(* CODESYS project Rasi_feeds_batching2.project

Project tree, tasks and I/O mapping:
  PLC_AC500_V3 : PM5032-T-ETH, ABB AG, order no. 1SAP123400R0x72, version 3.7.0.0
    application Application
      libraries: ModbusRtu, * (ABB); Util, * (System)
      task Task (cyclic, interval t#10ms, priority 14, watchdog t#20ms x 1) calls batching14
      CheckConfigurationObject
      Diagnosis/
        text list Diag_IO_Bus
        text list Diag_V3_PLC
      global variables GVL
      function block Auto_Batching_V14 [ST]
      function block Semi_Auto_Batching_V14 [ST]
      program batching14 [FBD]
      function block FB_Samyak_Multi [ST]
      function block FB_Samyak_Control [ST]
    OnBoard_IO : 12DI/8DO-T/2DC, ABB AG, version 3.7.0.0
        input  E_Stop_DI : BOOL  // Fast inputs DI0-DI3.Digital input DI0
        input  Run_PB : BOOL  // Fast inputs DI0-DI3.Digital input DI1
        unmapped channels: Fast inputs DI0-DI3, Fast inputs DI4-DI7, Standard inputs DI8-DI11, Digital inputs - Transistor, Fast outputs DO0-DO3, Fast outputs DO4-DO7, Digital outputs - Transistor
    IO_Bus : I/O-Bus, ABB AG, version 3.7.0.0
    Interfaces : Interfaces, ABB AG, version 3.7.0.0
      TA5142_RS485I : TA5142-RS485I, ABB AG, order no. 1SAP187300R0x02, version 3.7.0.0
        Modbus_RTU_Client : Modbus RTU Client, ABB AG, version 3.7.0.0
      OptionSlot_2
      Ethernet : Ethernet, ABB AG, version 3.7.0.0
        ETH1 : IP Settings, ABB AG, version 3.7.0.0
          NetConfig : NetConfig, ABB AG, version 3.7.0.0
          Modbus_TCP_IP_Server : Modbus TCP/IP Server, ABB AG, version 3.7.0.0
        Protocols : Client Protocols, ABB AG, version 3.7.0.0
    OnBoard_RTC : OnBoard RTC, ABB AG, version 3.7.0.0
  text list GlobalTextList
*)

// PLC_AC500_V3/Application/GVL
{attribute 'qualified_only'}
VAR_GLOBAL
    Recipe_Weights AT %MD100 : ARRAY[1..20] OF REAL;
	Auto_Bin_Material_Mapping AT %MW50: ARRAY[1..6] OF INT;
	Semi_Auto_Bin_Material_Mapping AT %MW60: ARRAY[1..10] OF INT;
	Auto_Coarse_To_Fine_speed AT %MD120: ARRAY[1..6] OF REAL := [1.0,1.0,1.0,1.0,1.0,1.0];
	Semi_Auto_Coarse_To_Fine_speed AT %MD130: ARRAY[1..10] OF REAL := [1.0,1.0,1.0,1.0,1.0,1.0,1.0,1.0,1.0,1.0];
	Auto_Bin_Tolerance AT %MD150: ARRAY[1..6] OF REAL;
	Semi_Auto_Bin_Tolerance AT %MD160: ARRAY[1..10] OF REAL;
	Start_Button AT %MX2.0: BOOL;
	E_Stop_Active AT %MX2.1: BOOL;
	Reset AT %MX2.3: BOOL;
	Next_Cycle_Start AT %MX2.4: BOOL;               // Command pulse/signal to start next batch cycle after hoppers are emptied
	Auto_Active_Mat AT %MW70: INT;
	Auto_Active_Bin AT %MW71: INT;
	Semi_Auto_Active_Mat AT %MW72: INT;
	Semi_Auto_Active_Bin AT %MW73: INT;
	Target_Batch_Cycles AT %MW74: INT := 1;
	Current_Batch_Cycle AT %MW75: INT;
	Completed_Batch_Cycles AT %MW79: INT;
	Error_Code AT %MW76: INT;
	Run AT %MX2.5 : BOOL;
	load_cell_auto AT %MD174 : REAL;
	load_cell_semi_auto AT %MD175 : REAL;
	Auto_Initial_Tolerance AT %MD176 : REAL := 5.0;
	Semi_Auto_Initial_Tolerance AT %MD178 : REAL := 5.0;
	Empty_Weight_Limit AT %MD186 : REAL := 5.0;     // Maximum scale weight limit (kg) to qualify scale as empty before starting next cycle
	Auto_Total_Target_Weight AT %MD170 : REAL;
	Semi_Auto_Total_Target_Weight AT %MD171 : REAL;
	Auto_Material_Count AT %MW77: INT;
	Semi_Auto_Material_Count AT %MW78 : INT;
	Auto_Current_Step AT %MW80 : INT;
	Semi_Auto_Current_Step AT %MW81 : INT;
	Auto_Active_Target_Weight AT %MD220 : REAL;
	Semi_Auto_Active_Target_Weight AT %MD224 : REAL;
	Auto_Active_Live_Weight AT %MD172 : REAL;
	Semi_Auto_Active_Live_Weight AT %MD173 : REAL;
	Auto_Excess_Allowed AT %MX2.6 : BOOL;
	Semi_Auto_Excess_Allowed AT %MX2.9 : BOOL;
	Auto_Excess_Alarm AT %MX2.7 : BOOL;
	Semi_Auto_Excess_Alarm AT %MX2.8 : BOOL;
	Auto_Inter_Bin_Delay AT %MD190 : TIME;
	Semi_Auto_Inter_Bin_Delay AT %MD194 : TIME;
	Auto_Sequence_Complete AT %MX3.0 : BOOL;
	Semi_Auto_Sequence_Complete AT %MX3.1 : BOOL;
	All_Cycles_Complete AT %MX3.2 : BOOL;           // Master flag: TRUE when all target batch cycles have completed
	Auto_Status_Message : STRING(80);
	Semi_Auto_Status_Message : STRING(80);
	
	(* 8 Process Output and Weight Arrays *)
	Auto_Bin : ARRAY[1..6] OF BOOL;
	auto_bin_cutoff : ARRAY[1..6] OF BOOL;
	auto_bin_motor : ARRAY[1..6] OF BOOL;
	Semi_Auto_Bin : ARRAY[1..10] OF BOOL;
	semi_auto_bin_cutoff : ARRAY[1..10] OF BOOL;
	semi_auto_bin_motor : ARRAY[1..10] OF BOOL;
	Auto_Weights : ARRAY[1..6] OF REAL;
	Semi_Auto_Weights : ARRAY[1..10] OF REAL;
END_VAR

// PLC_AC500_V3/Application/batching14
PROGRAM batching14
VAR
	Auto_Ctrl: Auto_Batching_V14;
	Semi_Auto_Ctrl: Semi_Auto_Batching_V14;
	Auto_Complete: BOOL;
	Semi_Auto_Complete: BOOL;
	Auto_Err: INT;
	Auto_Msg: STRING;
	Semi_Auto_Err: INT;
	Semi_Auto_Msg: STRING;
	AutoBatchScale: MODRTUMAST;
	ModEnabler: BLINK;
	SamyakRaw: ARRAY[0..1] OF DINT;
	AutBatchRaw: ARRAY[0..1] OF DINT;
	SemAutoScale: MODRTUMAST;
	SemiAutoScaleRaw: ARRAY[0..1] OF DINT;
	AutoBatchSamyak: REAL;
	FB_Samyak_Multi_1: FB_Samyak_Multi;
	
	FB_Samyak_Control_1: FB_Samyak_Control;
	Run_PB_1: BOOL;
	Next_Cycle_Start: BOOL;
END_VAR

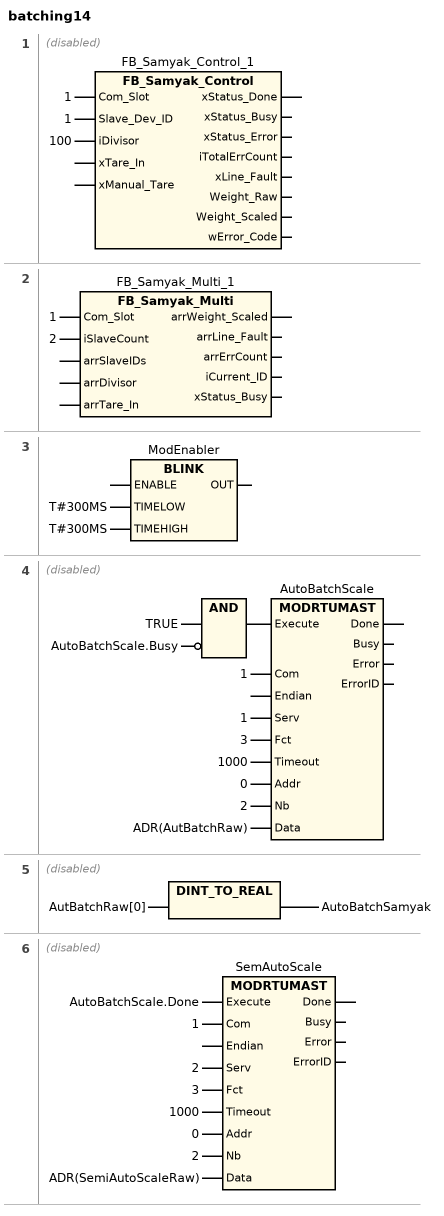
// NETWORK 1 (disabled)
// FB_Samyak_Control_1(Com_Slot := 1, Slave_Dev_ID := 1, iDivisor := 100); // FB_Samyak_Control

// NETWORK 2
FB_Samyak_Multi_1(Com_Slot := 1, iSlaveCount := 2); // FB_Samyak_Multi

// NETWORK 3
ModEnabler(TIMELOW := T#300MS, TIMEHIGH := T#300MS); // BLINK

// NETWORK 4 (disabled)
// AutoBatchScale(
//     Execute := TRUE AND NOT AutoBatchScale.Busy,
//     Com := 1,
//     Serv := 1,
//     Fct := 3,
//     Timeout := 1000,
//     Addr := 0,
//     Nb := 2,
//     Data := ADR(AutBatchRaw)); // MODRTUMAST

// NETWORK 5 (disabled)
// AutoBatchSamyak := DINT_TO_REAL(AutBatchRaw[0]);

// NETWORK 6 (disabled)
// SemAutoScale(
//     Execute := AutoBatchScale.Done,
//     Com := 1,
//     Serv := 2,
//     Fct := 3,
//     Timeout := 1000,
//     Addr := 0,
//     Nb := 2,
//     Data := ADR(SemiAutoScaleRaw)); // MODRTUMAST

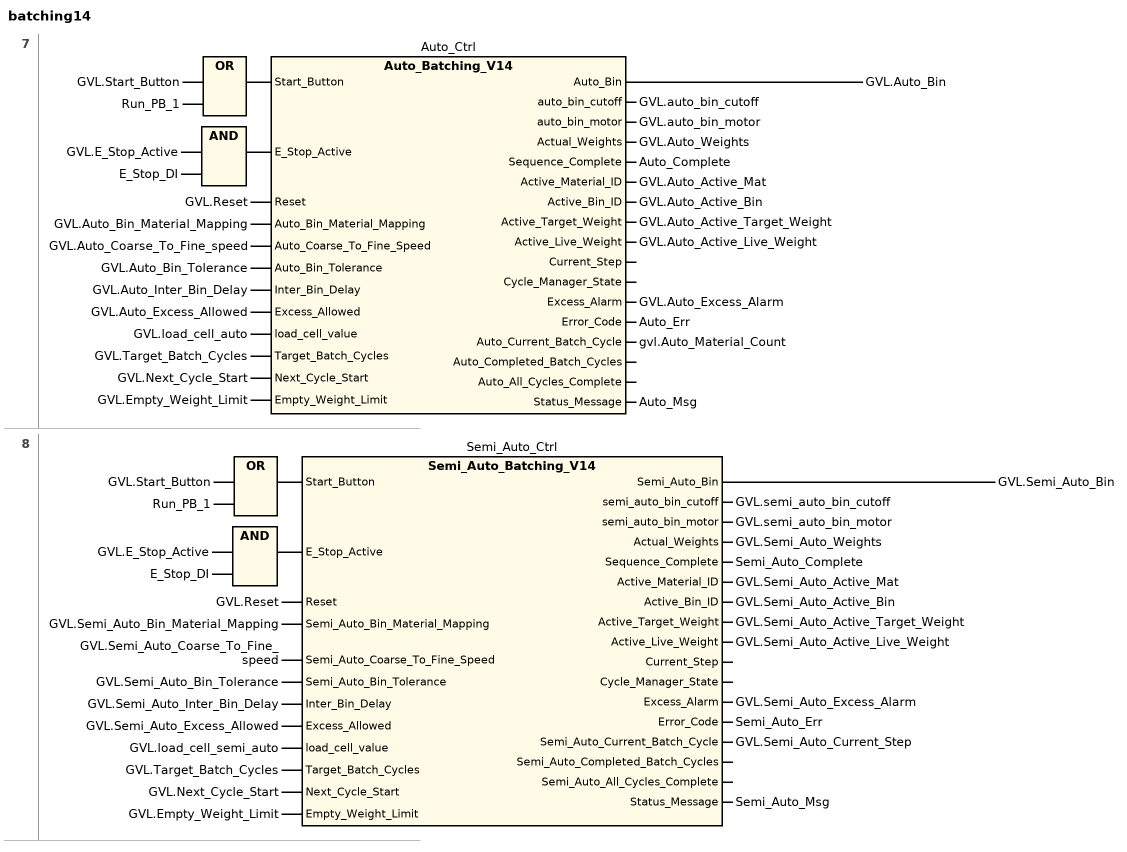
// NETWORK 7
Auto_Ctrl(
    Start_Button := GVL.Start_Button OR Run_PB_1,
    E_Stop_Active := GVL.E_Stop_Active AND E_Stop_DI,
    Reset := GVL.Reset,
    Auto_Bin_Material_Mapping := GVL.Auto_Bin_Material_Mapping,
    Auto_Coarse_To_Fine_Speed := GVL.Auto_Coarse_To_Fine_speed,
    Auto_Bin_Tolerance := GVL.Auto_Bin_Tolerance,
    Inter_Bin_Delay := GVL.Auto_Inter_Bin_Delay,
    Excess_Allowed := GVL.Auto_Excess_Allowed,
    load_cell_value := GVL.load_cell_auto,
    Target_Batch_Cycles := GVL.Target_Batch_Cycles,
    Next_Cycle_Start := GVL.Next_Cycle_Start,
    Empty_Weight_Limit := GVL.Empty_Weight_Limit,
    auto_bin_cutoff => GVL.auto_bin_cutoff,
    auto_bin_motor => GVL.auto_bin_motor,
    Actual_Weights => GVL.Auto_Weights,
    Sequence_Complete => Auto_Complete,
    Active_Material_ID => GVL.Auto_Active_Mat,
    Active_Bin_ID => GVL.Auto_Active_Bin,
    Active_Target_Weight => GVL.Auto_Active_Target_Weight,
    Active_Live_Weight => GVL.Auto_Active_Live_Weight,
    Excess_Alarm => GVL.Auto_Excess_Alarm,
    Error_Code => Auto_Err,
    Auto_Current_Batch_Cycle => gvl.Auto_Material_Count,
    Status_Message => Auto_Msg); // Auto_Batching_V14
GVL.Auto_Bin := Auto_Ctrl.Auto_Bin;

// NETWORK 8
Semi_Auto_Ctrl(
    Start_Button := GVL.Start_Button OR Run_PB_1,
    E_Stop_Active := GVL.E_Stop_Active AND E_Stop_DI,
    Reset := GVL.Reset,
    Semi_Auto_Bin_Material_Mapping := GVL.Semi_Auto_Bin_Material_Mapping,
    Semi_Auto_Coarse_To_Fine_Speed := GVL.Semi_Auto_Coarse_To_Fine_speed,
    Semi_Auto_Bin_Tolerance := GVL.Semi_Auto_Bin_Tolerance,
    Inter_Bin_Delay := GVL.Semi_Auto_Inter_Bin_Delay,
    Excess_Allowed := GVL.Semi_Auto_Excess_Allowed,
    load_cell_value := GVL.load_cell_semi_auto,
    Target_Batch_Cycles := GVL.Target_Batch_Cycles,
    Next_Cycle_Start := GVL.Next_Cycle_Start,
    Empty_Weight_Limit := GVL.Empty_Weight_Limit,
    semi_auto_bin_cutoff => GVL.semi_auto_bin_cutoff,
    semi_auto_bin_motor => GVL.semi_auto_bin_motor,
    Actual_Weights => GVL.Semi_Auto_Weights,
    Sequence_Complete => Semi_Auto_Complete,
    Active_Material_ID => GVL.Semi_Auto_Active_Mat,
    Active_Bin_ID => GVL.Semi_Auto_Active_Bin,
    Active_Target_Weight => GVL.Semi_Auto_Active_Target_Weight,
    Active_Live_Weight => GVL.Semi_Auto_Active_Live_Weight,
    Excess_Alarm => GVL.Semi_Auto_Excess_Alarm,
    Error_Code => Semi_Auto_Err,
    Semi_Auto_Current_Batch_Cycle => GVL.Semi_Auto_Current_Step,
    Status_Message => Semi_Auto_Msg); // Semi_Auto_Batching_V14
GVL.Semi_Auto_Bin := Semi_Auto_Ctrl.Semi_Auto_Bin;

END_PROGRAM

// PLC_AC500_V3/Application/FB_Samyak_Control
FUNCTION_BLOCK FB_Samyak_Control
VAR_INPUT
    Com_Slot      : BYTE := 1;     (* PLC COM port *)
    Slave_Dev_ID  : BYTE := 1;     (* Samyak slave ID *)
    iDivisor      : REAL := 10.0;  (* Scale factor: Weight_Scaled = Raw / iDivisor *)
    xTare_In      : BOOL;           (* Logic tare pulse *)
    xManual_Tare  : BOOL;           (* HMI/manual tare pulse *)
END_VAR

VAR_OUTPUT
    xStatus_Done   : BOOL;
    xStatus_Busy   : BOOL;
    xStatus_Error  : BOOL;
    iTotalErrCount : INT := 0;
    xLine_Fault    : BOOL;
    Weight_Raw     : DINT;
    Weight_Scaled  : REAL;
    wError_Code    : WORD; (* Check PLC & SAMYAK BaudRate, DevId, Parity; also check PLC serial port LED blink status and RS485 connection if error repeats *)
END_VAR

VAR
    fbRead         : ModRtuMast;
    fbTare         : ModRtuMast;
    iStep          : INT := 0;
    Samyak_Buffer  : ARRAY[0..17] OF WORD;
    wTareCommand   : WORD := 1;

    rtTareTrig     : R_TRIG;
    rtErrTrig      : R_TRIG;
    tStuckWatchdog : TON;
    tRecoveryTimer : TON;

    xTareReq       : BOOL := FALSE; (* Internal tare request latch *)
END_VAR


(* --- 1) Error Tracking + Auto Recovery --- *)
tStuckWatchdog(IN := (fbRead.Busy OR fbTare.Busy), PT := T#2000MS);

rtErrTrig(CLK := (fbRead.Error OR fbTare.Error));
IF rtErrTrig.Q THEN
    iTotalErrCount := iTotalErrCount + 1;
END_IF

IF fbRead.Done OR fbTare.Done THEN
    iTotalErrCount := 0;
    xLine_Fault := FALSE;
END_IF

IF iTotalErrCount >= 10 THEN
    xLine_Fault := TRUE;
END_IF

tRecoveryTimer(IN := xLine_Fault, PT := T#5S);
IF tRecoveryTimer.Q THEN
    iTotalErrCount := 0;
    xLine_Fault := FALSE;
END_IF

IF tStuckWatchdog.Q THEN
    iStep := 99;
END_IF

(* Capture tare request from either input pulse *)
rtTareTrig(CLK := xTare_In OR xManual_Tare);
IF rtTareTrig.Q THEN
    xTareReq := TRUE;
END_IF

(* --- 2) Modbus State Machine --- *)
CASE iStep OF

    0:  (* Continuous Read *)
        fbTare(Execute := FALSE);

        fbRead(
            Execute := NOT (fbRead.Done OR fbRead.Error OR fbRead.Busy)
                       AND NOT xTareReq
                       AND NOT xLine_Fault,
            COM     := Com_Slot,
            Serv    := Slave_Dev_ID,
            FCT     := 3,
            Addr    := 0,
            Nb      := 2,
            Data    := ADR(Samyak_Buffer[0]),
            Timeout := 400,
            Done    => xStatus_Done,
            Busy    => xStatus_Busy,
            Error   => xStatus_Error,
            ErrorID => wError_Code
        );

        IF xStatus_Done THEN
            Weight_Raw := TO_DINT(SHL(TO_DWORD(Samyak_Buffer[1]), 16) OR TO_DWORD(Samyak_Buffer[0]));
            Weight_Scaled := TO_REAL(Weight_Raw) / iDivisor;
        END_IF

        IF xTareReq THEN
            iStep := 1;
        END_IF

    1:  (* Port Release *)
        fbRead(Execute := FALSE);
        IF NOT fbRead.Busy THEN
            iStep := 2;
        END_IF

    2:  (* Execute Tare *)
        fbTare(
            Execute := TRUE,
            COM     := Com_Slot,
            Serv    := Slave_Dev_ID,
            FCT     := 6,
            Addr    := 16,
            Nb      := 1,
            Data    := ADR(wTareCommand),
            Timeout := 1000,
            Done    => xStatus_Done,
            Busy    => xStatus_Busy,
            Error   => xStatus_Error,
            ErrorID => wError_Code
        );

        IF fbTare.Done OR fbTare.Error THEN
            xTareReq := FALSE;
            iStep := 3;
        END_IF

    3:  (* Return to Read *)
        fbTare(Execute := FALSE);
        IF NOT fbTare.Busy THEN
            iStep := 0;
        END_IF

    99: (* Emergency Recovery *)
        fbRead(Execute := FALSE);
        fbTare(Execute := FALSE);

        IF NOT (fbRead.Busy OR fbTare.Busy) THEN
            iTotalErrCount := 0;
            iStep := 0;
        END_IF

END_CASE

END_FUNCTION_BLOCK

// PLC_AC500_V3/Application/FB_Samyak_Multi
//SAMYAK 4016 Multi Slave Unit Customised Block
//Note: This FB_Samyak_Multi name is impotrtant when you create new POU.

FUNCTION_BLOCK FB_Samyak_Multi
VAR_INPUT
    Com_Slot      : BYTE := 1;    (* Port Number *)
    iSlaveCount   : INT := 1;     (* How many slaves active: 1 to 4 *)
    arrSlaveIDs   : ARRAY[1..4] OF BYTE := [1, 2, 3, 4]; (* Unit IDs *)
    arrDivisor    : ARRAY[1..4] OF REAL := [10.0, 10.0, 10.0, 10.0]; (* Scaling per Unit *)
    arrTare_In    : ARRAY[1..4] OF BOOL; (* Individual Tare triggers *)
END_VAR

VAR_OUTPUT
    arrWeight_Scaled : ARRAY[1..4] OF REAL; (* Scaled result per unit *)
    arrLine_Fault    : ARRAY[1..4] OF BOOL; (* Fault status per unit *)
    arrErrCount      : ARRAY[1..4] OF INT;  (* Error count per unit *)
    iCurrent_ID      : BYTE;                (* Current ID being polled *)
    xStatus_Busy     : BOOL;                (* Overall Bus Busy *)
END_VAR

VAR
    (* Internal ModRtuMast Instances *)
    fbRead         : ModRtuMast;
    fbTare         : ModRtuMast;
    
    (* Polling Control *)
    iStep          : INT := 0;
    iIdx           : INT := 1;    (* Current Loop Index *)
    Samyak_Buffer  : ARRAY[0..17] OF WORD;
    wTareCommand   : WORD := 1;
    
    (* Unique Timer/Trigger Instances *)
    rtTareTrig     : R_TRIG;
    rtErrTrig      : R_TRIG;
    tWatchdog      : TON;
    tRecovery      : TON;
END_VAR



(* --- 1. INDIVIDUAL UNIT MONITORING --- *)
iCurrent_ID := arrSlaveIDs[iIdx]; 

(* Watchdog for Bus Hangs *)
tWatchdog(IN := (fbRead.Busy OR fbTare.Busy), PT := T#2000MS);
xStatus_Busy := fbRead.Busy OR fbTare.Busy;

(* Error Tracking for Current Index *)
rtErrTrig(CLK := (fbRead.Error OR fbTare.Error));
IF rtErrTrig.Q THEN
    arrErrCount[iIdx] := arrErrCount[iIdx] + 1;
END_IF

(* Reset on Success *)
IF fbRead.Done OR fbTare.Done THEN
    arrErrCount[iIdx] := 0;
    arrLine_Fault[iIdx] := FALSE;
END_IF

(* Line Fault Activation (10 errors) *)
IF arrErrCount[iIdx] >= 10 THEN
    arrLine_Fault[iIdx] := TRUE;
END_IF

(* Auto-Recovery pulse (5s) *)
tRecovery(IN := arrLine_Fault[iIdx], PT := T#5S);
IF tRecovery.Q THEN
    arrErrCount[iIdx] := 0;
    arrLine_Fault[iIdx] := FALSE;
END_IF

IF tWatchdog.Q THEN iStep := 99; END_IF

(* Check Tare for active slave *)
rtTareTrig(CLK := arrTare_In[iIdx]);

(* --- 2. SEQUENTIAL STATE MACHINE --- *)
CASE iStep OF
    
    0: (* READ CURRENT SLAVE *)
        fbTare(Execute := FALSE);
        fbRead(
            Execute := NOT (fbRead.Done OR fbRead.Error OR fbRead.Busy) 
                       AND NOT rtTareTrig.Q AND NOT arrLine_Fault[iIdx],
            COM     := Com_Slot,
            Serv    := arrSlaveIDs[iIdx],
            FCT     := 3, Addr := 0, Nb := 2, 
            Data    := ADR(Samyak_Buffer[0]), Timeout := 400
        );

        IF fbRead.Done THEN
            (* Scale weight using the array-based divisor for this specific index *)
            arrWeight_Scaled[iIdx] := TO_REAL(TO_DINT(SHL(TO_DWORD(Samyak_Buffer[1]), 16) OR TO_DWORD(Samyak_Buffer[0]))) / arrDivisor[iIdx];
            iStep := 10; (* Switch to next slave *)
        END_IF
        
        IF fbRead.Error THEN iStep := 10; END_IF (* Move on if error *)
        IF rtTareTrig.Q THEN iStep := 1; END_IF  (* Priority: Tare current unit *)

    1: (* PORT RELEASE *)
        fbRead(Execute := FALSE);
        IF NOT fbRead.Busy THEN iStep := 2; END_IF

    2: (* WRITE TARE FOR CURRENT SLAVE *)
        fbTare(
            Execute := TRUE,
            COM := Com_Slot, Serv := arrSlaveIDs[iIdx], 
            FCT := 6, Addr := 16, Nb := 1,
            Data := ADR(wTareCommand), Timeout := 1000
        );

        IF fbTare.Done OR fbTare.Error THEN
            arrTare_In[iIdx] := FALSE; (* Reset manual trigger *)
            iStep := 3;
        END_IF

    3: (* CLEANUP *)
        fbTare(Execute := FALSE);
        IF NOT fbTare.Busy THEN iStep := 10; END_IF

    10: (* INDEX ROTATION *)
        iIdx := iIdx + 1;
        IF iIdx > iSlaveCount THEN
            iIdx := 1; (* Back to first slave *)
        END_IF
        iStep := 0;

    99: (* EMERGENCY RESET *)
        fbRead(Execute := FALSE); fbTare(Execute := FALSE);
        IF NOT (fbRead.Busy OR fbTare.Busy) THEN iStep := 0; END_IF
        
END_CASE

END_FUNCTION_BLOCK

// PLC_AC500_V3/Application/Auto_Batching_V14
FUNCTION_BLOCK Auto_Batching_V14
VAR_INPUT
    Start_Button : BOOL;                            // Command pulse/signal to start or resume the auto batching sequence
    E_Stop_Active : BOOL;                           // Emergency Stop circuit status (NC contact: TRUE = Healthy/Run permitted, FALSE = E-Stop tripped)
    Reset : BOOL;                                   // System reset pulse (clears active steps, outputs, alarms, and error flags)
    Auto_Bin_Material_Mapping : ARRAY[1..6] OF INT; // Array mapping physical Silos 1..6 to Recipe Material IDs (1..20, 0 = Silo skipped)
    Auto_Coarse_To_Fine_Speed : ARRAY[1..6] OF REAL;// Weight offset threshold (kg) before target to transition from Coarse to Fine feeding
    Auto_Bin_Tolerance : ARRAY[1..6] OF REAL;       // Allowable weight tolerance window (±kg) around target weight for each silo
    Inter_Bin_Delay : TIME;                         // Settling delay duration after completing a bin before advancing to the next
    Excess_Allowed : BOOL;                          // Overfill handling policy: TRUE = proceed if target is exceeded, FALSE = raise alarm and halt
    load_cell_value : REAL;                         // Live gross weight input reading from the Auto scale load cell (kg)
    Target_Batch_Cycles : INT;                      // Target number of batch cycle repetitions configured from HMI (defaults to 1)
    Next_Cycle_Start : BOOL;                        // Command pulse/signal to start next batch cycle after hoppers are emptied
    Empty_Weight_Limit : REAL;                      // Maximum scale weight limit (kg) for scales to qualify as empty before starting next cycle
END_VAR
VAR_OUTPUT
    Auto_Bin : ARRAY[1..6] OF BOOL;                 // Coarse feeding valve / gate actuation command outputs for Silos 1..6
    auto_bin_cutoff : ARRAY[1..6] OF BOOL;          // Fine feeding valve / vibrator cutoff actuation command outputs for Silos 1..6
    auto_bin_motor : ARRAY[1..6] OF BOOL;           // Feeder / screw conveyor motor run commands for Silos 1..6
    Actual_Weights : ARRAY[1..6] OF REAL;           // Net material weight (kg) successfully dosed for each silo in the current cycle
    Sequence_Complete : BOOL;                       // Handshake flag: TRUE when all mapped Auto silos have completed dosing and settling
    Active_Material_ID : INT;                       // Recipe Material ID currently being dosed (1..20, 0 when idle/complete)
    Active_Bin_ID : INT;                            // Physical Silo index currently being dosed (1..6, 0 when idle/complete)
    Active_Target_Weight : REAL;                    // Target weight setpoint (kg) of the ingredient currently being dosed
    Active_Live_Weight : REAL;                      // Live net/tared weight (kg) accumulated into the scale for the active silo
    Current_Step : INT;                             // Real-time sequence step:
                                                    //   0  = Idle / Waiting for Start
                                                    //   1..6 = Dosing Silos 1..6 (feeding coarse/fine)
                                                    //   7  = Settling delay in progress
                                                    //   8  = Sequence complete
    Cycle_Manager_State : INT;                      // Master supervisory cycle manager state:
                                                    //   0  = System Idle / Stopped
                                                    //   1  = Running active batch cycle
                                                    //   4  = All target batch cycles completed successfully
                                                    //   5  = Paused between cycles (Cycle Hold active)
    Excess_Alarm : BOOL;                            // Overfill alarm: TRUE when dosed weight exceeds target + tolerance (with Excess_Allowed=FALSE)
    Error_Code : INT;                               // Fault diagnostic code:
                                                    //   0  = No Error / System Healthy
                                                    //   1  = Duplicate Material ID mapped across Auto and Semi-Auto
                                                    //   2  = Material index out of range (must be 1..20)
                                                    //   3  = Recipe weight is less than (Coarse_To_Fine_Speed + Tolerance)
                                                    //   4  = Initial scale tare error (scale not empty before start)
                                                    //   21 = Scale overload protection triggered (> 500 kg)
    Auto_Current_Batch_Cycle : INT;                     // Active batch cycle number currently processing (1..Target_Batch_Cycles)
    Auto_Completed_Batch_Cycles : INT;                  // Total number of batch cycle loops completed successfully
    Auto_All_Cycles_Complete : BOOL;                    // Master flag: TRUE when all Target_Batch_Cycles have finished
    Status_Message : STRING(80);                    // Real-time human-readable process status and diagnostic text message
END_VAR
VAR
    bin_last_weight : REAL;
    actual_bin : REAL;
    target_weight : REAL;
    cutoff_trigger_weight : REAL;
    min_tol_weight : REAL;
    max_tol_weight : REAL;
    Paused_By_EStop : BOOL;
    Effective_Delay : TIME;
    Mat_Idx : INT;
    i : INT;
    j : INT;
    Transition_Timer : TON;
    Completion_Timer : TON;
    Simulation_Mode : BOOL;
    Sim_Rate : REAL;
    Sim_Timer : TON;
    Start_Sim_Weight : REAL;
    Discharge_Active : BOOL;
    
    (* Master Cycle Manager & Supervisory states *)
    Internal_FB_Start : BOOL;
    Duplicate_Found : BOOL;
    Invalid_Material_Range : BOOL;
    Weight_Limit_Error : BOOL;
    eff_empty_limit : REAL;
    Next_Cycle_Last : BOOL;
    Next_Cycle_Rising : BOOL;
END_VAR


(* Auto Batching FB V14 with Full Diagnostics, Step Tracking, and Precise Status Reporting *)

Effective_Delay := Inter_Bin_Delay;
IF Effective_Delay = T#0S THEN
    Effective_Delay := T#2S;
END_IF;

(* Detect rising edge on Next_Cycle_Start trigger *)
Next_Cycle_Rising := (Next_Cycle_Start OR GVL.Next_Cycle_Start) AND NOT Next_Cycle_Last;
Next_Cycle_Last := (Next_Cycle_Start OR GVL.Next_Cycle_Start);

(* 1. RECIPE TOTALS & SUPERVISORY CONFIGURATION CHECKS *)
Duplicate_Found := FALSE;
Invalid_Material_Range := FALSE;
Weight_Limit_Error := FALSE;

GVL.Auto_Total_Target_Weight := 0.0;
GVL.Auto_Material_Count := 0;
FOR i := 1 TO 6 DO
    IF Auto_Bin_Material_Mapping[i] < 0 OR Auto_Bin_Material_Mapping[i] > 20 THEN
        Invalid_Material_Range := TRUE;
    END_IF;
    IF Auto_Bin_Material_Mapping[i] <> 0 AND Auto_Bin_Material_Mapping[i] <= 20 THEN
        FOR j := 1 TO 10 DO
            IF Auto_Bin_Material_Mapping[i] = GVL.Semi_Auto_Bin_Material_Mapping[j] THEN
                Duplicate_Found := TRUE;
            END_IF;
        END_FOR;
    END_IF;
    IF Auto_Bin_Material_Mapping[i] > 0 AND Auto_Bin_Material_Mapping[i] <= 20 THEN
        IF GVL.Recipe_Weights[Auto_Bin_Material_Mapping[i]] > 0.0 THEN
            GVL.Auto_Total_Target_Weight := GVL.Auto_Total_Target_Weight + GVL.Recipe_Weights[Auto_Bin_Material_Mapping[i]];
            GVL.Auto_Material_Count := GVL.Auto_Material_Count + 1;
            IF GVL.Recipe_Weights[Auto_Bin_Material_Mapping[i]] < (Auto_Coarse_To_Fine_Speed[i] + Auto_Bin_Tolerance[i]) THEN
                Weight_Limit_Error := TRUE;
            END_IF;
        END_IF;
    END_IF;
END_FOR;

IF Duplicate_Found THEN
    GVL.Error_Code := 1;
    Error_Code := 1;
    Status_Message := 'Error 1: Duplicate Material ID mapped in Auto and Semi-Auto!';
ELSIF Invalid_Material_Range THEN
    GVL.Error_Code := 2;
    Error_Code := 2;
    Status_Message := 'Error 2: Material Index configuration out of range (1..20)!';
ELSIF Weight_Limit_Error THEN
    GVL.Error_Code := 3;
    Error_Code := 3;
    Status_Message := 'Error 3: Recipe weight is less than Coarse_To_Fine_Speed + Tolerance!';
ELSE
    IF GVL.Error_Code <= 3 THEN
        GVL.Error_Code := 0;
        Error_Code := 0;
    END_IF;
END_IF;

(* 2. HARD RESET INTERLOCK *)
IF Reset OR GVL.Reset THEN
    FOR i := 1 TO 6 DO
        Auto_Bin[i] := FALSE;
        auto_bin_cutoff[i] := FALSE;
        auto_bin_motor[i] := FALSE;
        Actual_Weights[i] := 0.0;
        GVL.Auto_Bin[i] := FALSE;
        GVL.auto_bin_cutoff[i] := FALSE;
        GVL.auto_bin_motor[i] := FALSE;
        GVL.Auto_Weights[i] := 0.0;
    END_FOR;
    
    (* Reset Recipe & Active Target Setpoints *)
    FOR i := 1 TO 20 DO
        GVL.Recipe_Weights[i] := 0.0;
    END_FOR;
    GVL.Auto_Total_Target_Weight := 0.0;
    GVL.Semi_Auto_Total_Target_Weight := 0.0;
    GVL.Auto_Material_Count := 0;
    GVL.Semi_Auto_Material_Count := 0;
    
    Sequence_Complete := FALSE;
    GVL.Auto_Sequence_Complete := FALSE;
    GVL.Semi_Auto_Sequence_Complete := FALSE;
    Active_Material_ID := 0;
    Active_Bin_ID := 0;
    Active_Target_Weight := 0.0;
    Active_Live_Weight := 0.0;
    GVL.Auto_Active_Target_Weight := 0.0;
    GVL.Auto_Active_Live_Weight := 0.0;
    Excess_Alarm := FALSE;
    Error_Code := 0;
    GVL.Error_Code := 0;
    GVL.Current_Batch_Cycle := 0;
    GVL.Completed_Batch_Cycles := 0;
    GVL.All_Cycles_Complete := FALSE;
    Auto_Completed_Batch_Cycles := 0;
    Auto_Current_Batch_Cycle := 0;
    Auto_All_Cycles_Complete := FALSE;
    GVL.Target_Batch_Cycles := 0;
    GVL.Start_Button := FALSE;
    GVL.Run := FALSE;
    GVL.Next_Cycle_Start := FALSE;
    Next_Cycle_Last := FALSE;
    Next_Cycle_Rising := FALSE;
    GVL.Auto_Active_Mat := 0;
    GVL.Auto_Active_Bin := 0;
    GVL.Auto_Excess_Alarm := FALSE;
    Current_Step := 0;
    Cycle_Manager_State := 0;
    Internal_FB_Start := FALSE;
    bin_last_weight := 0.0;
    Start_Sim_Weight := 0.0;
    Transition_Timer(IN := FALSE);
    Completion_Timer(IN := FALSE);
    Sim_Timer(IN := FALSE);
    Status_Message := 'Auto [Reset]: System Reset Complete - System Idle';
    RETURN;
END_IF;

(* 3. E-STOP PAUSE / HOLD LOGIC (NC Contact: FALSE = Pressed/Tripped, TRUE = Healthy) *)
IF NOT E_Stop_Active OR NOT GVL.E_Stop_Active THEN
    Paused_By_EStop := TRUE;
END_IF;

IF Paused_By_EStop THEN
    FOR i := 1 TO 6 DO
        Auto_Bin[i] := FALSE;
        auto_bin_cutoff[i] := FALSE;
        auto_bin_motor[i] := FALSE;
    END_FOR;
    IF NOT E_Stop_Active OR NOT GVL.E_Stop_Active THEN
        Status_Message := CONCAT('Auto [PAUSED]: E-Stop Active at Step ', INT_TO_STRING(Current_Step));
    ELSE
        Status_Message := CONCAT('Auto [HOLD]: E-Stop Cleared. Press Start to Resume Step ', INT_TO_STRING(Current_Step));
        IF Start_Button OR GVL.Start_Button THEN
            Paused_By_EStop := FALSE;
        END_IF;
    END_IF;
    Sim_Timer(IN := FALSE);
    Transition_Timer(IN := FALSE);
    Completion_Timer(IN := FALSE);
    RETURN;
END_IF;

(* 4. MASTER CYCLE MANAGER STATE MACHINE *)
CASE Cycle_Manager_State OF
    0: (* IDLE *)
        Internal_FB_Start := FALSE;
        GVL.Run := FALSE;
        GVL.Next_Cycle_Start := FALSE;
        GVL.Auto_Sequence_Complete := FALSE;
        
        IF GVL.Error_Code = 0 AND NOT (Start_Button OR GVL.Start_Button) THEN
            Status_Message := 'Auto [State 0 - Idle]: Ready - Waiting for Start Button';
        END_IF;
        
        IF Start_Button OR GVL.Start_Button THEN
            (* Use Target_Batch_Cycles from input, or fallback to GVL, or default to 1 *)
            IF Target_Batch_Cycles > 0 THEN
                GVL.Target_Batch_Cycles := Target_Batch_Cycles;
            ELSIF GVL.Target_Batch_Cycles <= 0 THEN
                GVL.Target_Batch_Cycles := 1;
            END_IF;
            
            IF NOT E_Stop_Active OR NOT GVL.E_Stop_Active THEN
                GVL.Run := FALSE;
                Status_Message := 'Auto [State 0]: Cannot Start - Emergency Stop Contact Open!';
            ELSIF (GVL.Auto_Initial_Tolerance > 0.0 AND (GVL.load_cell_auto > GVL.Auto_Initial_Tolerance OR GVL.load_cell_auto < (-GVL.Auto_Initial_Tolerance))) OR 
                  (GVL.Semi_Auto_Initial_Tolerance > 0.0 AND (GVL.load_cell_semi_auto > GVL.Semi_Auto_Initial_Tolerance OR GVL.load_cell_semi_auto < (-GVL.Semi_Auto_Initial_Tolerance))) THEN
                GVL.Run := FALSE;
                GVL.Error_Code := 4;
                Error_Code := 4;
                Status_Message := 'Auto [State 0]: Error 4 - Scale not zeroed (exceeds Initial Tolerance)!';
            ELSE
                GVL.Error_Code := 0;
                Error_Code := 0;
                GVL.Current_Batch_Cycle := 1;
                GVL.Completed_Batch_Cycles := 0;
                GVL.All_Cycles_Complete := FALSE;
                Auto_Completed_Batch_Cycles := 0;
                Auto_Current_Batch_Cycle := 1;
                Auto_All_Cycles_Complete := FALSE;
                GVL.Run := TRUE;
                Internal_FB_Start := TRUE;
                Cycle_Manager_State := 1;
                Current_Step := 0;
            END_IF;
        END_IF;
        
    1: (* RUNNING CYCLE *)
        Internal_FB_Start := TRUE;
        GVL.Run := TRUE;
        
        (* Interlock: While process is actively running, Next_Cycle_Start MUST be FALSE *)
        GVL.Next_Cycle_Start := FALSE;
        
        (* Both Auto and Semi-Auto must complete to finish the cycle *)
        IF Sequence_Complete AND GVL.Semi_Auto_Sequence_Complete THEN
            GVL.Completed_Batch_Cycles := GVL.Current_Batch_Cycle;
            Auto_Completed_Batch_Cycles := GVL.Current_Batch_Cycle;
            IF GVL.Current_Batch_Cycle < GVL.Target_Batch_Cycles AND GVL.Error_Code = 0 THEN
                Internal_FB_Start := FALSE;
                Cycle_Manager_State := 5; (* Go to pause/hold to wait for scale empty & Next_Cycle_Start *)
            ELSE
                Cycle_Manager_State := 4; (* All target cycles completed *)
            END_IF;
        END_IF;
        
    5: (* PAUSED BETWEEN CYCLES - WAITING FOR HOPPERS EMPTIED & NEXT CYCLE START *)
        Internal_FB_Start := FALSE;
        GVL.Run := TRUE;
        
        (* Determine effective empty weight threshold (defaults to 5.0 kg if <= 0.0) *)
        eff_empty_limit := Empty_Weight_Limit;
        IF eff_empty_limit <= 0.0 THEN
            eff_empty_limit := GVL.Empty_Weight_Limit;
        END_IF;
        IF eff_empty_limit <= 0.0 THEN
            eff_empty_limit := 5.0;
        END_IF;
        
        Status_Message := CONCAT('Auto [State 5]: Cycle ', CONCAT(INT_TO_STRING(GVL.Current_Batch_Cycle), ' Done. Empty scales < limit and trigger Next_Cycle_Start.'));
        
        (* Check ONLY on a new trigger pulse (rising edge) of Next_Cycle_Start *)
        IF Next_Cycle_Rising THEN
            (* Check both scales are below the empty weight limit at the moment of trigger *)
            IF (GVL.load_cell_auto < eff_empty_limit) AND (GVL.load_cell_semi_auto < eff_empty_limit) THEN
                (* Scale is empty: momentary reset of command, advance to next cycle *)
                GVL.Next_Cycle_Start := FALSE;
                Next_Cycle_Last := FALSE;
                GVL.Start_Button := TRUE; (* Keep Start_Button TRUE until all cycles are complete! *)
                GVL.Error_Code := 0;
                Error_Code := 0;
                GVL.Current_Batch_Cycle := GVL.Current_Batch_Cycle + 1;
                Auto_Current_Batch_Cycle := GVL.Current_Batch_Cycle;
                Sequence_Complete := FALSE;
                GVL.Auto_Sequence_Complete := FALSE;
                GVL.Semi_Auto_Sequence_Complete := FALSE;
                Current_Step := 0;
                Internal_FB_Start := TRUE;
                Cycle_Manager_State := 1;
                FOR i := 1 TO 6 DO
                    Actual_Weights[i] := 0.0;
                    Auto_Bin[i] := FALSE;
                    auto_bin_cutoff[i] := FALSE;
                    auto_bin_motor[i] := FALSE;
                END_FOR;
            ELSE
                (* Scale not empty yet: reject trigger, reset command, and wait for operator to trigger again *)
                GVL.Next_Cycle_Start := FALSE;
                Next_Cycle_Last := FALSE;
                Status_Message := CONCAT('Auto [State 5]: Scale weight exceeds limit (', CONCAT(REAL_TO_STRING(eff_empty_limit), ' kg)! Empty scales and trigger Next_Cycle_Start again.'));
            END_IF;
        END_IF;
        
    4: (* ALL CYCLES COMPLETE *)
        Internal_FB_Start := FALSE;
        GVL.Run := FALSE;
        GVL.Start_Button := FALSE;
        Auto_All_Cycles_Complete := TRUE;
        GVL.All_Cycles_Complete := TRUE;
        Sequence_Complete := TRUE;
        GVL.Auto_Sequence_Complete := TRUE;
        GVL.Semi_Auto_Sequence_Complete := TRUE;
        Status_Message := CONCAT('Auto [State 4 - Finished]: All ', CONCAT(INT_TO_STRING(GVL.Target_Batch_Cycles), ' Batch Cycles Completed Successfully'));
        IF Start_Button OR GVL.Start_Button THEN
            (* Reset flags for new batch start *)
            Current_Step := 0;
            Auto_All_Cycles_Complete := FALSE;
            GVL.All_Cycles_Complete := FALSE;
            Sequence_Complete := FALSE;
            GVL.Auto_Sequence_Complete := FALSE;
            GVL.Semi_Auto_Sequence_Complete := FALSE;
            Cycle_Manager_State := 0;
        END_IF;
END_CASE;

(* 5. AUTO SILOS 1..6 POURING SEQUENCE WITH DETAILED STATUS *)
IF Current_Step = 0 AND Internal_FB_Start THEN
    Current_Step := 1;
    bin_last_weight := load_cell_value;
    Sequence_Complete := FALSE;
    GVL.Auto_Sequence_Complete := FALSE;
    Excess_Alarm := FALSE;
    Error_Code := 0;
    FOR i := 1 TO 6 DO
        Actual_Weights[i] := 0.0;
        Auto_Bin[i] := FALSE;
        auto_bin_cutoff[i] := FALSE;
        auto_bin_motor[i] := FALSE;
    END_FOR;
END_IF;

CASE Current_Step OF
    0:
        Active_Material_ID := 0;
        Active_Bin_ID := 0;
        Excess_Alarm := FALSE;
        Sequence_Complete := FALSE;
        FOR i := 1 TO 6 DO
            Auto_Bin[i] := FALSE;
            auto_bin_cutoff[i] := FALSE;
            auto_bin_motor[i] := FALSE;
        END_FOR;
        Active_Target_Weight := GVL.Auto_Active_Target_Weight;
        Active_Live_Weight := 0.0;
        
    1..6:
        (* Skip any bin where Material Mapping is 0, > 20, or Recipe Weight is 0 *)
        WHILE Current_Step >= 1 AND Current_Step <= 6 DO
            Mat_Idx := Auto_Bin_Material_Mapping[Current_Step];
            IF Mat_Idx = 0 OR Mat_Idx > 20 OR GVL.Recipe_Weights[Mat_Idx] <= 0.0 THEN
                Auto_Bin[Current_Step] := FALSE;
                auto_bin_cutoff[Current_Step] := FALSE;
                auto_bin_motor[Current_Step] := FALSE;
                Actual_Weights[Current_Step] := 0.0;
                IF Current_Step = 6 THEN
                    Current_Step := 7;
                    EXIT;
                ELSE
                    Current_Step := Current_Step + 1;
                END_IF;
            ELSE
                EXIT; (* Valid active recipe silo found *)
            END_IF;
        END_WHILE;
        
        IF Current_Step = 7 THEN
            Active_Material_ID := 0;
            Active_Bin_ID := 0;
            Active_Target_Weight := 0.0;
            Active_Live_Weight := 0.0;
            GVL.Auto_Active_Target_Weight := 0.0;
            GVL.Auto_Active_Live_Weight := 0.0;
            Status_Message := 'Auto [Step 7]: Settling Delay in progress...';
            Completion_Timer(IN := TRUE, PT := Effective_Delay);
            IF Completion_Timer.Q THEN
                Completion_Timer(IN := FALSE);
                Current_Step := 8;
            END_IF;
        ELSE
            Mat_Idx := Auto_Bin_Material_Mapping[Current_Step];
            target_weight := GVL.Recipe_Weights[Mat_Idx];
            
            Active_Target_Weight := target_weight;
            GVL.Auto_Active_Target_Weight := target_weight;
            
            cutoff_trigger_weight := target_weight - Auto_Coarse_To_Fine_Speed[Current_Step];
            min_tol_weight := target_weight - Auto_Bin_Tolerance[Current_Step];
            max_tol_weight := target_weight + Auto_Bin_Tolerance[Current_Step];
            
            actual_bin := load_cell_value - bin_last_weight;
            IF actual_bin < 0.0 THEN
                actual_bin := 0.0;
            END_IF;
            Actual_Weights[Current_Step] := actual_bin;
            Active_Live_Weight := actual_bin;
            GVL.Auto_Active_Live_Weight := actual_bin;
            Active_Material_ID := Mat_Idx;
            Active_Bin_ID := Current_Step;
            
            IF load_cell_value > 500.0 THEN
                Error_Code := 21;
                GVL.Error_Code := 21;
                Status_Message := CONCAT('Auto [Step ', CONCAT(INT_TO_STRING(Current_Step), ']: STUCK - Error 21: Scale Overloaded (> 500 kg)!'));
                Sequence_Complete := TRUE;
                GVL.Auto_Sequence_Complete := TRUE;
                Paused_By_EStop := TRUE;
            END_IF;
            
            IF actual_bin < cutoff_trigger_weight THEN
                Auto_Bin[Current_Step] := TRUE;
                auto_bin_cutoff[Current_Step] := FALSE;
                auto_bin_motor[Current_Step] := TRUE;
                Excess_Alarm := FALSE;
                Status_Message := CONCAT('Auto [Step ', CONCAT(INT_TO_STRING(Current_Step), ']: Coarse Feeding'));
            ELSIF actual_bin < min_tol_weight THEN
                Auto_Bin[Current_Step] := FALSE;
                auto_bin_cutoff[Current_Step] := TRUE;
                auto_bin_motor[Current_Step] := TRUE;
                Excess_Alarm := FALSE;
                Status_Message := CONCAT('Auto [Step ', CONCAT(INT_TO_STRING(Current_Step), ']: Fine Feeding'));
            ELSIF actual_bin > max_tol_weight THEN
                Auto_Bin[Current_Step] := FALSE;
                auto_bin_cutoff[Current_Step] := FALSE;
                auto_bin_motor[Current_Step] := FALSE;
                IF Excess_Allowed THEN
                    Excess_Alarm := FALSE;
                    Status_Message := CONCAT('Auto [Step ', CONCAT(INT_TO_STRING(Current_Step), ']: Excess Allowed - Advancing'));
                    bin_last_weight := load_cell_value;
                    Active_Target_Weight := 0.0;
                    Active_Live_Weight := 0.0;
                    GVL.Auto_Active_Target_Weight := 0.0;
                    GVL.Auto_Active_Live_Weight := 0.0;
                    IF Current_Step = 6 THEN
                        Current_Step := 7;
                    ELSE
                        Current_Step := Current_Step + 1;
                    END_IF;
                ELSE
                    Excess_Alarm := TRUE;
                    Status_Message := CONCAT('Auto [Step ', CONCAT(INT_TO_STRING(Current_Step), ']: STUCK - Excess Weight! Reduce weight or enable Excess Allowed.'));
                END_IF;
            ELSE
                Auto_Bin[Current_Step] := FALSE;
                auto_bin_cutoff[Current_Step] := FALSE;
                auto_bin_motor[Current_Step] := FALSE;
                Excess_Alarm := FALSE;
                bin_last_weight := load_cell_value;
                Active_Target_Weight := 0.0;
                Active_Live_Weight := 0.0;
                GVL.Auto_Active_Target_Weight := 0.0;
                GVL.Auto_Active_Live_Weight := 0.0;
                Status_Message := CONCAT('Auto [Step ', CONCAT(INT_TO_STRING(Current_Step), ']: Target Reached - Advancing'));
                IF Current_Step = 6 THEN
                    Current_Step := 7;
                ELSE
                    Current_Step := Current_Step + 1;
                END_IF;
            END_IF;
        END_IF;

    7:
        Active_Material_ID := 0;
        Active_Bin_ID := 0;
        Excess_Alarm := FALSE;
        Status_Message := 'Auto [Step 7]: Settling Delay in progress...';
        Completion_Timer(IN := TRUE, PT := Effective_Delay);
        IF Completion_Timer.Q THEN
            Completion_Timer(IN := FALSE);
            Current_Step := 8;
        END_IF;
        
    8:
        Active_Material_ID := 0;
        Active_Bin_ID := 0;
        Excess_Alarm := FALSE;
        Sequence_Complete := TRUE;
        GVL.Auto_Sequence_Complete := TRUE;
        IF NOT GVL.Semi_Auto_Sequence_Complete THEN
            Status_Message := 'Auto [Step 8]: Auto Finished. Waiting for Semi-Auto to complete...';
        ELSE
            Status_Message := 'Auto [Step 8]: Cycle Sequences Complete';
        END_IF;
END_CASE;

(* Synchronize physical output arrays to GVL *)
FOR i := 1 TO 6 DO
    GVL.Auto_Bin[i] := Auto_Bin[i];
    GVL.auto_bin_cutoff[i] := auto_bin_cutoff[i];
    GVL.auto_bin_motor[i] := auto_bin_motor[i];
END_FOR;

(* Synchronize live cycle progress to outputs *)
Auto_Current_Batch_Cycle := GVL.Current_Batch_Cycle;
Auto_Completed_Batch_Cycles := GVL.Completed_Batch_Cycles;
Auto_All_Cycles_Complete := GVL.All_Cycles_Complete;

END_FUNCTION_BLOCK

// PLC_AC500_V3/Application/Semi_Auto_Batching_V14
FUNCTION_BLOCK Semi_Auto_Batching_V14
VAR_INPUT
    Start_Button : BOOL;                                 // Command pulse/signal to start or resume the semi-auto batching sequence
    E_Stop_Active : BOOL;                                // Emergency Stop circuit status (NC contact: TRUE = Healthy/Run permitted, FALSE = E-Stop tripped)
    Reset : BOOL;                                        // System reset pulse (clears active steps, outputs, alarms, and error flags)
    Semi_Auto_Bin_Material_Mapping : ARRAY[1..10] OF INT;// Array mapping physical Silos 1..10 to Recipe Material IDs (1..20, 0 = Silo skipped)
    Semi_Auto_Coarse_To_Fine_Speed : ARRAY[1..10] OF REAL;// Weight offset threshold (kg) before target to transition from Coarse to Fine feeding
    Semi_Auto_Bin_Tolerance : ARRAY[1..10] OF REAL;      // Allowable weight tolerance window (±kg) around target weight for each silo
    Inter_Bin_Delay : TIME;                              // Settling delay duration after completing a bin before advancing to the next
    Excess_Allowed : BOOL;                               // Overfill handling policy: TRUE = proceed if target is exceeded, FALSE = raise alarm and halt
    load_cell_value : REAL;                              // Live gross weight input reading from the Semi-Auto scale load cell (kg)
    Target_Batch_Cycles : INT;                           // Target number of batch cycle repetitions configured from HMI (defaults to 1)
    Next_Cycle_Start : BOOL;                             // Command pulse/signal to start next batch cycle after hoppers are emptied
    Empty_Weight_Limit : REAL;                           // Maximum scale weight limit (kg) for scales to qualify as empty before starting next cycle
END_VAR
VAR_OUTPUT
    Semi_Auto_Bin : ARRAY[1..10] OF BOOL;                // Coarse feeding valve / gate actuation command outputs for Silos 1..10
    semi_auto_bin_cutoff : ARRAY[1..10] OF BOOL;         // Fine feeding valve / vibrator cutoff actuation command outputs for Silos 1..10
    semi_auto_bin_motor : ARRAY[1..10] OF BOOL;          // Feeder / screw conveyor motor run commands for Silos 1..10
    Actual_Weights : ARRAY[1..10] OF REAL;               // Net material weight (kg) successfully dosed for each silo in the current cycle
    Sequence_Complete : BOOL;                            // Handshake flag: TRUE when all mapped Semi-Auto silos have completed dosing and settling
    Active_Material_ID : INT;                            // Recipe Material ID currently being dosed (1..20, 0 when idle/complete)
    Active_Bin_ID : INT;                                 // Physical Silo index currently being dosed (1..10, 0 when idle/complete)
    Active_Target_Weight : REAL;                         // Target weight setpoint (kg) of the ingredient currently being dosed
    Active_Live_Weight : REAL;                           // Live net/tared weight (kg) accumulated into the scale for the active silo
    Current_Step : INT;                                  // Real-time sequence step:
                                                         //   0   = Idle / Waiting for Start
                                                         //   1..10 = Dosing Silos 1..10 (feeding coarse/fine)
                                                         //   31  = Settling delay in progress
                                                         //   32  = Sequence complete
    Cycle_Manager_State : INT;                           // Master supervisory cycle manager state:
                                                         //   0   = System Idle / Stopped
                                                         //   1   = Running active batch cycle
                                                         //   4   = All target batch cycles completed successfully
                                                         //   5   = Paused between cycles (Cycle Hold active)
    Excess_Alarm : BOOL;                                 // Overfill alarm: TRUE when dosed weight exceeds target + tolerance (with Excess_Allowed=FALSE)
    Error_Code : INT;                                    // Fault diagnostic code:
                                                         //   0   = No Error / System Healthy
                                                         //   1   = Duplicate Material ID mapped across Auto and Semi-Auto
                                                         //   2   = Material index out of range (must be 1..20)
                                                         //   3   = Recipe weight is less than (Coarse_To_Fine_Speed + Tolerance)
                                                         //   4   = Initial scale tare error (scale not empty before start)
                                                         //   21  = Scale overload protection triggered (> 500 kg)
    Semi_Auto_Current_Batch_Cycle : INT;                 // Active batch cycle number currently processing (1..Target_Batch_Cycles)
    Semi_Auto_Completed_Batch_Cycles : INT;              // Total number of batch cycle loops completed successfully
    Semi_Auto_All_Cycles_Complete : BOOL;                // Master flag: TRUE when all Target_Batch_Cycles have finished
    Status_Message : STRING(80);                         // Real-time human-readable process status and diagnostic text message
END_VAR
VAR
    bin_last_weight : REAL;
    actual_bin : REAL;
    target_weight : REAL;
    cutoff_trigger_weight : REAL;
    min_tol_weight : REAL;
    max_tol_weight : REAL;
    Paused_By_EStop : BOOL;
    Effective_Delay : TIME;
    Mat_Idx : INT;
    i : INT;
    Last_Batch_Cycle : INT;
    Transition_Timer : TON;
    Completion_Timer : TON;
    Simulation_Mode : BOOL;
    Sim_Rate : REAL;
    Sim_Timer : TON;
    Start_Sim_Weight : REAL;
    Discharge_Active : BOOL;
    Run_Last : BOOL;
    Run_Rising : BOOL;
END_VAR


(* Semi-Auto Batching FB V14 with Full Diagnostics, Step Tracking, and Precise Status Reporting *)

Effective_Delay := Inter_Bin_Delay;
IF Effective_Delay = T#0S THEN
    Effective_Delay := T#2S;
END_IF;

(* Track Master Cycle State *)
IF Target_Batch_Cycles > 0 THEN
    GVL.Target_Batch_Cycles := Target_Batch_Cycles;
END_IF;

(* Master Cycle State & Start Synchronization *)
Run_Rising := GVL.Run AND NOT Run_Last;
Run_Last := GVL.Run;

IF GVL.Run THEN
    IF Sequence_Complete AND GVL.Auto_Sequence_Complete THEN
        IF GVL.Current_Batch_Cycle >= GVL.Target_Batch_Cycles AND GVL.Target_Batch_Cycles > 0 THEN
            Cycle_Manager_State := 4;
        ELSE
            Cycle_Manager_State := 5;
        END_IF;
    ELSE
        Cycle_Manager_State := 1;
    END_IF;
ELSE
    Cycle_Manager_State := 0;
    Current_Step := 0;
    Last_Batch_Cycle := 0;
    Sequence_Complete := FALSE;
    GVL.Semi_Auto_Sequence_Complete := FALSE;
END_IF;

(* On fresh batch start (rising edge of Run), ensure clean start from Step 0 *)
IF Run_Rising THEN
    Current_Step := 0;
    Last_Batch_Cycle := 0;
    Sequence_Complete := FALSE;
    GVL.Semi_Auto_Sequence_Complete := FALSE;
END_IF;

(* 1. SEMI-AUTO RECIPE TOTALS & ACTIVE SILO COUNT *)
GVL.Semi_Auto_Total_Target_Weight := 0.0;
GVL.Semi_Auto_Material_Count := 0;
FOR i := 1 TO 10 DO
    IF Semi_Auto_Bin_Material_Mapping[i] > 0 AND Semi_Auto_Bin_Material_Mapping[i] <= 20 THEN
        IF GVL.Recipe_Weights[Semi_Auto_Bin_Material_Mapping[i]] > 0.0 THEN
            GVL.Semi_Auto_Total_Target_Weight := GVL.Semi_Auto_Total_Target_Weight + GVL.Recipe_Weights[Semi_Auto_Bin_Material_Mapping[i]];
            GVL.Semi_Auto_Material_Count := GVL.Semi_Auto_Material_Count + 1;
        END_IF;
    END_IF;
END_FOR;

(* 2. HARD RESET INTERLOCK *)
IF Reset OR GVL.Reset THEN
    FOR i := 1 TO 10 DO
        Semi_Auto_Bin[i] := FALSE;
        semi_auto_bin_cutoff[i] := FALSE;
        semi_auto_bin_motor[i] := FALSE;
        Actual_Weights[i] := 0.0;
        GVL.Semi_Auto_Bin[i] := FALSE;
        GVL.semi_auto_bin_cutoff[i] := FALSE;
        GVL.semi_auto_bin_motor[i] := FALSE;
        GVL.Semi_Auto_Weights[i] := 0.0;
    END_FOR;
    Sequence_Complete := FALSE;
    GVL.Semi_Auto_Sequence_Complete := FALSE;
    Active_Material_ID := 0;
    Active_Bin_ID := 0;
    Active_Target_Weight := 0.0;
    Active_Live_Weight := 0.0;
    GVL.Semi_Auto_Active_Target_Weight := 0.0;
    GVL.Semi_Auto_Active_Live_Weight := 0.0;
    GVL.Semi_Auto_Active_Mat := 0;
    GVL.Semi_Auto_Active_Bin := 0;
    GVL.Semi_Auto_Excess_Alarm := FALSE;
    Excess_Alarm := FALSE;
    Error_Code := 0;
    Paused_By_EStop := FALSE;
    Current_Step := 0;
    Last_Batch_Cycle := 0;
    Cycle_Manager_State := 0;
    Semi_Auto_Current_Batch_Cycle := 0;
    Semi_Auto_Completed_Batch_Cycles := 0;
    Semi_Auto_All_Cycles_Complete := FALSE;
    bin_last_weight := 0.0;
    Start_Sim_Weight := 0.0;
    Run_Last := FALSE;
    Run_Rising := FALSE;
    Transition_Timer(IN := FALSE);
    Completion_Timer(IN := FALSE);
    Sim_Timer(IN := FALSE);
    Status_Message := 'Semi-Auto [Reset]: System Reset Complete - System Idle';
    
    (* Clean Auto-Clearing: Reset has been processed by both blocks *)
    GVL.Reset := FALSE;
    RETURN;
END_IF;

(* 3. E-STOP PAUSE / HOLD LOGIC (NC Contact: FALSE = Pressed/Tripped, TRUE = Healthy) *)
IF NOT E_Stop_Active OR NOT GVL.E_Stop_Active THEN
    Paused_By_EStop := TRUE;
END_IF;

IF Paused_By_EStop THEN
    FOR i := 1 TO 10 DO
        Semi_Auto_Bin[i] := FALSE;
        semi_auto_bin_cutoff[i] := FALSE;
        semi_auto_bin_motor[i] := FALSE;
    END_FOR;
    IF NOT E_Stop_Active OR NOT GVL.E_Stop_Active THEN
        Status_Message := CONCAT('Semi-Auto [PAUSED]: E-Stop Active at Step ', INT_TO_STRING(Current_Step));
    ELSE
        Status_Message := CONCAT('Semi-Auto [HOLD]: E-Stop Cleared. Press Start to Resume Step ', INT_TO_STRING(Current_Step));
        IF Start_Button OR GVL.Start_Button THEN
            Paused_By_EStop := FALSE;
        END_IF;
    END_IF;
    Sim_Timer(IN := FALSE);
    Transition_Timer(IN := FALSE);
    Completion_Timer(IN := FALSE);
    RETURN;
END_IF;

(* 4. CYCLE COMPLETE / HOLD STATE *)
IF Cycle_Manager_State = 5 THEN
    Status_Message := 'Semi-Auto [Cycle Complete]: Waiting for scale empty & Next_Cycle_Start...';
END_IF;

(* 5. SEQUENCE START (FOR CYCLE 1 AND REPEAT CYCLES) *)
IF GVL.Run AND Cycle_Manager_State <> 5 THEN
    IF Current_Step = 0 THEN
        (* Initial cycle start *)
        Last_Batch_Cycle := GVL.Current_Batch_Cycle;
        Current_Step := 1;
        bin_last_weight := load_cell_value;
        Sequence_Complete := FALSE;
        GVL.Semi_Auto_Sequence_Complete := FALSE;
        Excess_Alarm := FALSE;
        Error_Code := 0;
        FOR i := 1 TO 10 DO
            Actual_Weights[i] := 0.0;
            Semi_Auto_Bin[i] := FALSE;
            semi_auto_bin_cutoff[i] := FALSE;
            semi_auto_bin_motor[i] := FALSE;
        END_FOR;
    ELSIF Current_Step = 32 AND GVL.Current_Batch_Cycle <> Last_Batch_Cycle THEN
        (* Advance to next cycle loop (Cycle 2, 3, etc.) *)
        Last_Batch_Cycle := GVL.Current_Batch_Cycle;
        Current_Step := 1;
        bin_last_weight := load_cell_value;
        Sequence_Complete := FALSE;
        GVL.Semi_Auto_Sequence_Complete := FALSE;
        Excess_Alarm := FALSE;
        Error_Code := 0;
        FOR i := 1 TO 10 DO
            Actual_Weights[i] := 0.0;
            Semi_Auto_Bin[i] := FALSE;
            semi_auto_bin_cutoff[i] := FALSE;
            semi_auto_bin_motor[i] := FALSE;
        END_FOR;
    END_IF;
END_IF;

CASE Current_Step OF
    0:
        Active_Material_ID := 0;
        Active_Bin_ID := 0;
        Excess_Alarm := FALSE;
        Sequence_Complete := FALSE;
        FOR i := 1 TO 10 DO
            Semi_Auto_Bin[i] := FALSE;
            semi_auto_bin_cutoff[i] := FALSE;
            semi_auto_bin_motor[i] := FALSE;
        END_FOR;
        Active_Target_Weight := GVL.Semi_Auto_Active_Target_Weight;
        Active_Live_Weight := 0.0;
        IF Error_Code = 0 AND Cycle_Manager_State <> 5 THEN 
            Status_Message := 'Semi-Auto [Step 0 - Idle]: Ready - Waiting for Run Signal'; 
        END_IF;
        
    1..10:
        (* Skip any bin where Material Mapping is 0, > 20, or Recipe Weight is 0 *)
        WHILE Current_Step >= 1 AND Current_Step <= 10 DO
            Mat_Idx := Semi_Auto_Bin_Material_Mapping[Current_Step];
            IF Mat_Idx = 0 OR Mat_Idx > 20 OR GVL.Recipe_Weights[Mat_Idx] <= 0.0 THEN
                Semi_Auto_Bin[Current_Step] := FALSE;
                semi_auto_bin_cutoff[Current_Step] := FALSE;
                semi_auto_bin_motor[Current_Step] := FALSE;
                Actual_Weights[Current_Step] := 0.0;
                IF Current_Step = 10 THEN
                    Current_Step := 31;
                    EXIT;
                ELSE
                    Current_Step := Current_Step + 1;
                END_IF;
            ELSE
                EXIT; (* Valid active recipe silo found *)
            END_IF;
        END_WHILE;
        
        IF Current_Step = 31 THEN
            Active_Material_ID := 0;
            Active_Bin_ID := 0;
            Active_Target_Weight := 0.0;
            Active_Live_Weight := 0.0;
            GVL.Semi_Auto_Active_Target_Weight := 0.0;
            GVL.Semi_Auto_Active_Live_Weight := 0.0;
            Status_Message := 'Semi-Auto [Step 31]: Settling Delay in progress...';
            Completion_Timer(IN := TRUE, PT := Effective_Delay);
            IF Completion_Timer.Q THEN
                Completion_Timer(IN := FALSE);
                Current_Step := 32;
            END_IF;
        ELSE
            Mat_Idx := Semi_Auto_Bin_Material_Mapping[Current_Step];
            target_weight := GVL.Recipe_Weights[Mat_Idx];
            
            Active_Target_Weight := target_weight;
            GVL.Semi_Auto_Active_Target_Weight := target_weight;
            
            cutoff_trigger_weight := target_weight - Semi_Auto_Coarse_To_Fine_Speed[Current_Step];
            min_tol_weight := target_weight - Semi_Auto_Bin_Tolerance[Current_Step];
            max_tol_weight := target_weight + Semi_Auto_Bin_Tolerance[Current_Step];
            
            actual_bin := load_cell_value - bin_last_weight;
            IF actual_bin < 0.0 THEN
                actual_bin := 0.0;
            END_IF;
            Actual_Weights[Current_Step] := actual_bin;
            Active_Live_Weight := actual_bin;
            GVL.Semi_Auto_Active_Live_Weight := actual_bin;
            Active_Material_ID := Mat_Idx;
            Active_Bin_ID := Current_Step;
            
            IF load_cell_value > 500.0 THEN
                Error_Code := 21;
                GVL.Error_Code := 21;
                Status_Message := CONCAT('Semi-Auto [Step ', CONCAT(INT_TO_STRING(Current_Step), ']: STUCK - Error 21: Scale Overloaded (> 500 kg)!'));
                Sequence_Complete := TRUE;
                GVL.Semi_Auto_Sequence_Complete := TRUE;
                Paused_By_EStop := TRUE;
            END_IF;
            
            IF actual_bin < cutoff_trigger_weight THEN
                Semi_Auto_Bin[Current_Step] := TRUE;
                semi_auto_bin_cutoff[Current_Step] := FALSE;
                semi_auto_bin_motor[Current_Step] := TRUE;
                Excess_Alarm := FALSE;
                Status_Message := CONCAT('Semi-Auto [Step ', CONCAT(INT_TO_STRING(Current_Step), ']: Coarse Feeding'));
            ELSIF actual_bin < min_tol_weight THEN
                Semi_Auto_Bin[Current_Step] := FALSE;
                semi_auto_bin_cutoff[Current_Step] := TRUE;
                semi_auto_bin_motor[Current_Step] := TRUE;
                Excess_Alarm := FALSE;
                Status_Message := CONCAT('Semi-Auto [Step ', CONCAT(INT_TO_STRING(Current_Step), ']: Fine Feeding'));
            ELSIF actual_bin > max_tol_weight THEN
                Semi_Auto_Bin[Current_Step] := FALSE;
                semi_auto_bin_cutoff[Current_Step] := FALSE;
                semi_auto_bin_motor[Current_Step] := FALSE;
                IF Excess_Allowed THEN
                    Excess_Alarm := FALSE;
                    Status_Message := CONCAT('Semi-Auto [Step ', CONCAT(INT_TO_STRING(Current_Step), ']: Excess Allowed - Advancing'));
                    bin_last_weight := load_cell_value;
                    Active_Target_Weight := 0.0;
                    Active_Live_Weight := 0.0;
                    GVL.Semi_Auto_Active_Target_Weight := 0.0;
                    GVL.Semi_Auto_Active_Live_Weight := 0.0;
                    IF Current_Step = 10 THEN
                        Current_Step := 31;
                    ELSE
                        Current_Step := Current_Step + 1;
                    END_IF;
                ELSE
                    Excess_Alarm := TRUE;
                    Status_Message := CONCAT('Semi-Auto [Step ', CONCAT(INT_TO_STRING(Current_Step), ']: STUCK - Excess Weight! Reduce weight or enable Excess Allowed.'));
                END_IF;
            ELSE
                Semi_Auto_Bin[Current_Step] := FALSE;
                semi_auto_bin_cutoff[Current_Step] := FALSE;
                semi_auto_bin_motor[Current_Step] := FALSE;
                Excess_Alarm := FALSE;
                bin_last_weight := load_cell_value;
                Active_Target_Weight := 0.0;
                Active_Live_Weight := 0.0;
                GVL.Semi_Auto_Active_Target_Weight := 0.0;
                GVL.Semi_Auto_Active_Live_Weight := 0.0;
                Status_Message := CONCAT('Semi-Auto [Step ', CONCAT(INT_TO_STRING(Current_Step), ']: Target Reached - Advancing'));
                IF Current_Step = 10 THEN
                    Current_Step := 31;
                ELSE
                    Current_Step := Current_Step + 1;
                END_IF;
            END_IF;
        END_IF;

    31:
        Active_Material_ID := 0;
        Active_Bin_ID := 0;
        Excess_Alarm := FALSE;
        Status_Message := 'Semi-Auto [Step 31]: Settling Delay in progress...';
        Completion_Timer(IN := TRUE, PT := Effective_Delay);
        IF Completion_Timer.Q THEN
            Completion_Timer(IN := FALSE);
            Current_Step := 32;
        END_IF;
        
    32:
        Active_Material_ID := 0;
        Active_Bin_ID := 0;
        Excess_Alarm := FALSE;
        Sequence_Complete := TRUE;
        GVL.Semi_Auto_Sequence_Complete := TRUE;
        IF NOT GVL.Auto_Sequence_Complete THEN
            Status_Message := 'Semi-Auto [Step 32]: Semi-Auto Finished. Waiting for Auto to complete...';
        ELSE
            Status_Message := 'Semi-Auto [Step 32]: Cycle Sequences Complete';
        END_IF;
END_CASE;

(* Synchronize physical output arrays to GVL *)
FOR i := 1 TO 10 DO
    GVL.Semi_Auto_Bin[i] := Semi_Auto_Bin[i];
    GVL.semi_auto_bin_cutoff[i] := semi_auto_bin_cutoff[i];
    GVL.semi_auto_bin_motor[i] := semi_auto_bin_motor[i];
END_FOR;

(* Synchronize live cycle progress to outputs *)
Semi_Auto_Current_Batch_Cycle := GVL.Current_Batch_Cycle;
Semi_Auto_Completed_Batch_Cycles := GVL.Completed_Batch_Cycles;
Semi_Auto_All_Cycles_Complete := GVL.All_Cycles_Complete;

END_FUNCTION_BLOCK

(* text list Diag_IO_Bus (id | default | en | de | fr | es | zh)
  Err_1037 | Test error | Test error | Testfehler |  |  | 测试错误
  Err_12 | Test pulse error -> Check wiring and sensor | Test pulse error -> Check wiring and sensor | Testimpuls-Fehler -> Verdrahtung und Sensor prüfen |  |  | 测试脉冲错误 -> 检查接线和传感器
  Err_13 | Test pulse cross-talk error -> Check wiring and sensor. If this error persists, replace I/O module. Contact ABB technical support. | Test pulse cross-talk error -> Check wiring and sensor. If this error persists, replace I/O module. Contact ABB technical support. | Fehler Testimpuls Kanalübersprechen  -> Verdrahtung und Sensor prüfen. Falls der Fehler weiterhin besteht, E/A-Modul austauschen. Technischen Support von ABB kontaktieren. |  |  | 测试脉冲串扰错误 -> 检查接线和传感器. 如果此错误仍然存在，请更换 I/O 模块. 联系 ABB 技术支持.
  Err_16128 | Failed max wait run | Failed max wait run | Lauf max. Warten fehlgeschlagen |  |  | 最大等待运行失败
  Err_16129 | Critical error, see log | Critical error, see log | Kritischer Fehler, siehe Protokoll |  |  | 严重错误，请参阅日志
  Err_16130 | Fatal error, see log | Fatal error, see log | Schwerwiegender Fehler, siehe Protokoll |  |  | 致命错误，请参阅日志
  Err_16131 | Timeout -> Replace I/O module | Timeout -> Replace I/O module | Timeout -> E/A-Modul austauschen |  |  | 超时 -> 更换 I/O 模块
  Err_16133 | Output data size mismatch | Output data size mismatch | Diskrepanz Ausgangsdatengröße |  |  | 输出数据大小不匹配
  Err_16134 | Input data size mismatch | Input data size mismatch | Diskrepanz Eingangsdatengröße |  |  | 输入数据大小不匹配
  Err_16137 | Overflow diagnosis buffer -> Restart | Overflow diagnosis buffer -> Restart | Überlauf Diagnosepuffer -> Neu Starten |  |  | 诊断缓冲区溢出 -> 重新启动
  Err_16138 | Non-safety I/O: Voltage overflow at outputs (above UP3 level), Safety I/O: Process voltage too high -> Check terminals / Check process voltage | Non-safety I/O: Voltage overflow at outputs (above UP3 level), Safety I/O: Process voltage too high -> Check terminals / Check process voltage | Standard-E/A: Spannungsüberlauf an Ausgängen (über UP3-Niveau), Sicherheits-E/A: Prozessspannung zu hoch -> Terminals prüfen / Prozessspannung prüfen |  |  | 非安全 I/O：输出端电压溢出（高于 UP3 电平），安全 I/O：过程电压过高 -> 检查终端 / 检查过程电压
  Err_16139 | Process voltage UP or UP3 too low -> Check process voltage | Process voltage UP or UP3 too low -> Check process voltage | Prozessspannung UP oder UP3 zu niedrig -> Prozessspannung prüfen |  |  | 过程电压 UP 或 UP3 过低 -> 检查过程电压
  Err_16145 | Error setting parameters | Error setting parameters | Fehlereinstellungsparameter |  |  | 设置参数时出错
  Err_16146 | Plausibility check failed (iParameter) -> Check configuration | Plausibility check failed (iParameter) -> Check configuration | Plausibilitätsprüfung fehlgeschlagen (iParameter) -> Konfiguration überprüfen |  |  | 合理性检查失败（i 参数） -> 检查配置
  Err_16147 | Checksum error -> Non-safety I/O: Replace I/O module. Safety I/O: Check safety configuration and CRCs for I- and F-Parameters. | Checksum error -> Non-safety I/O: Replace I/O module. Safety I/O: Check safety configuration and CRCs for I- and F-Parameters. | Prüfsummenfehler -> Standard-E/A: E/A-Modul austauschen. Sicherheits-E/A: Sicherheitskonfiguration und CRCs auf I- und F-Parameter prüfen. |  |  | 检校验和错误 -> 非安全 I/O：更换 I/O 模块. 安全 I/O：检查 I 参数和 F 参数的安全配置和 CRC.
  Err_16148 | PROFIsafe communication error -> Restart I/O module. If this error persists, contact ABB technical support. | PROFIsafe communication error -> Restart I/O module. If this error persists, contact ABB technical support. | PROFIsafe-Kommunikationsfehler -> E/A-Modul neu starten. Falls der Fehler weiterhin besteht, technischen Support von ABB kontaktieren. |  |  | PROFIsafe 通信错误 -> 重新启动 I/O 模块. 如果此错误仍然存在，请联系 ABB 技术支持.
  Err_16149 | No module data | No module data | Keine Moduldaten |  |  | 无模块数据
  Err_16153 | PROFIsafe watchdog timed out -> Restart I/O module. If this error persists, increase PROFIsafe watchdog time. | PROFIsafe watchdog timed out -> Restart I/O module. If this error persists, increase PROFIsafe watchdog time. | Timeout von PROFIsafe-Watchdog -> E/A-Modul neu starten. Falls der Fehler weiterhin besteht, PROFIsafe-Watchdog-Zeit verlängern. |  |  | PROFIsafe 看门狗超时 -> 重新启动 I/O 模块. 如果此错误仍然存在，请增加 PROFIsafe 看门狗时间.
  Err_16154 | Size of parameters expected by module differs from size provided by configuration -> Check master or configuration | Size of parameters expected by module differs from size provided by configuration -> Check master or configuration | Vom Modul erwartete Parametergröße weicht von der in der Konfiguration angegebenen Größe ab -> Master oder Konfiguration überprüfen |  |  | 模块期望的参数大小与配置提供的参数大小不同 -> 检查主设备或配置
  Err_16156 | F-Parameter configuration and address switch value do not match -> Check I/O module F-Parameter configuration and module address switch value. | F-Parameter configuration and address switch value do not match -> Check I/O module F-Parameter configuration and module address switch value. | Konfiguration für F-Parameter und Wert des Adressschalters stimmen nicht überein -> Konfiguration für F-Parameter des E/A-Moduls und Wert des Adressschalters überprüfen. |  |  | F 参数配置和地址开关值不匹配 -> 检查 I/O 模块 F 参数配置和模块地址开关值.
  Err_16158 | Type of present module does not match configuration | Type of present module does not match configuration | Typ des vorhandenen Moduls stimmt nicht mit Konfiguration überein |  |  | 当前模块类型与配置不匹配
  Err_16159 | Configured number of modules differs from found ones | Configured number of modules differs from found ones | Konfigurierte Anzahl von Modulen weicht von Anzahl gefundener Module ab |  |  | 配置的模块数量与找到的模块数量不同
  Err_16160 | At least one module failed during configuration | At least one module failed during configuration | Mindestens ein Modul während Konfiguration ausgefallen |  |  | 配置期间至少有一个模块发生故障
  Err_16164 | Internal data exchange failure -> Replace I/O module | Internal data exchange failure -> Replace I/O module | Fehler interner Datenaustausch -> E/A-Modul austauschen |  |  | 内部数据交换失败 -> 更换 I/O 模块
  Err_16168 | Different hard-/firmware versions in the module -> Replace I/O module | Different hard-/firmware versions in the module -> Replace I/O module | Unterschiedliche Hardware-/Firmware-Versionen im Modul -> E/A-Modul austauschen |  |  | 模块中的硬件/固件版本不同 -> 更换 I/O 模块
  Err_16171 | Internal error -> Replace I/O module | Internal error -> Replace I/O module | Interner Fehler -> E/A-Modul austauschen |  |  | 内部错误 -> 更换 I/O 模块
  Err_16172 | Has not passed factory test | Has not passed factory test | Hat Werksprüfung nicht bestanden |  |  | 未通过出厂测试
  Err_16173 | No process voltage UP or UP3 -> Check process voltage | No process voltage UP or UP3 -> Check process voltage | Keine Prozessspannung UP oder UP3 -> Prozessspannung prüfen |  |  | 无过程电压 UP 或 UP3 -> 检查过程电压
  Err_16175 | Sensor voltage too low | Sensor voltage too low | Sensorspannung zu niedrig |  |  | 传感器电压过低
  Err_16194 | Fatal error, not running any more | Fatal error, not running any more | Schwerwiegender Fehler, Ausführung gestoppt |  |  | 致命错误，不再运行
  Err_16246 | Failed to start the parameterization of modules | Failed to start the parameterization of modules | Starten von Parametrierung für Module fehlgeschlagen |  |  | 无法启动模块的参数化
  Err_16247 | Failed setting parameters | Failed setting parameters | Einstellen von Parametern fehlgeschlagen |  |  | 设置参数失败
  Err_16248 | Failed setting expected module | Failed setting expected module | Einstellen des erwarteten Moduls fehlgeschlagen |  |  | 设置预期模块失败
  Err_16254 | Size of parameters expected by module differs from size provided by configuration | Size of parameters expected by module differs from size provided by configuration | Vom Modul erwartete Parametergröße weicht von der in der Konfiguration angegebenen Größe ab |  |  | 模块期望的参数大小与配置提供的参数大小不同
  Err_18 | Test error | Test error | Testfehler |  |  | 测试错误
  Err_25 | Stuck at error -> Check I/O module wiring. Restart I/O module, if needed. If this error persists, replace I/O module. | Stuck at error -> Check I/O module wiring. Restart I/O module, if needed. If this error persists, replace I/O module. | Hängengeblieben bei Fehler -> Verdrahtung des E/A-Moduls überprüfen. Bei Bedarf E/A-Modul neu starten. Falls der Fehler weiterhin besteht, E/A-Modul austauschen. |  |  | 卡在错误处 -> 检查 I/O 模块接线. 如果需要，重新启动 I/O 模块. 如果此错误仍然存在，请更换 I/O 模块.
  Err_257 | Wrong measurement, false temperature at the compensation channel | Wrong measurement, false temperature at the compensation channel | Falscher Messwert, falsche Temperatur an Kompensationskanal |  |  | 测量值错误，补偿通道温度错误
  Err_258 | AI531: Wrong measurement; potential difference is too high; CD522: PWM duty cycle out of duty area | AI531: Wrong measurement; potential difference is too high; CD522: PWM duty cycle out of duty area | AI531: Falscher Messwert; Potenzialdifferenz zu hoch; CD522: PWM-Einschaltdauer außerhalb des Einschaltbereichs |  |  | AI531：测量错误; 电位差过高; CD522: PWM 占空比超出占空比范围
  Err_260 | Measurement overflow -> Check channel wiring and sensor power supply | Measurement overflow -> Check channel wiring and sensor power supply | Messwertüberschreitung -> Kanalverdrahtung und Spannungsversorgung des Sensors prüfen |  |  | 测量值溢出 -> 检查通道接线和传感器电源
  Err_263 | Measurement underflow -> Check channel wiring and sensor power supply | Measurement underflow -> Check channel wiring and sensor power supply | Messwertunterschreitung -> Kanalverdrahtung und Spannungsversorgung des Sensors prüfen |  |  | 测量值下溢 -> 检查通道接线和传感器电源
  Err_266 | Short circuit and cut wire or "out of range" | Short circuit and cut wire or "out of range" | Kurzschluss und Drahtbruch oder „außerhalb des zulässigen Bereichs“ |  |  | 短路和断线或“超出范围”
  Err_267 | Output/process voltage too low | Output/process voltage too low | Ausgangs-/Prozessspannung zu gering |  |  | 输出/过程电压过低
  Err_273 | Test error | Test error | Testfehler |  |  | 测试错误
  Err_28 | Cross-talk error -> Check I/O module wiring. Restart I/O module, if needed. If this error persists, replace I/O module. | Cross-talk error -> Check I/O module wiring. Restart I/O module, if needed. If this error persists, replace I/O module. | Fehler Kanalübersprechen -> Verdrahtung des E/A-Moduls überprüfen. Bei Bedarf E/A-Modul neu starten. Falls der Fehler weiterhin besteht, E/A-Modul austauschen. |  |  | 串扰错误 -> 检查 I/O 模块接线. 如果需要，重新启动 I/O 模块. 如果此错误仍然存在，请更换 I/O 模块.
  Err_3 | Discrepancy time expired -> Check discrepancy time value, channel wiring and sensor. | Discrepancy time expired -> Check discrepancy time value, channel wiring and sensor. | Diskrepanzzeit abgelaufen -> Diskrepanzzeit-Wert, Kanalverdrahtung und Sensor überprüfen. |  |  | 偏差时间已过 -> 检查差异时间值、通道接线和传感器.
  Err_303 | Short circuit at analog input -> Check channel wiring | Short circuit at analog input -> Check channel wiring | Kurzschluss an Analogeingang -> Kanalverdrahtung prüfen |  |  | 模拟输入端短路 -> 检查通道接线
  Err_304 | Analog value overflow or broken wire at an analog input -> Check value or check terminals | Analog value overflow or broken wire at an analog input -> Check value or check terminals | Analogwert-Überlauf oder Drahtbruch an Analogeingang -> Wert oder Terminals prüfen |  |  | 模拟输入端模拟值溢出或断线 -> 检查值或检查终端
  Err_311 | Value difference too high -> Adjust tolerance window for channels. Check channel wiring and sensor configuration. | Value difference too high -> Adjust tolerance window for channels. Check channel wiring and sensor configuration. | Wertdifferenz zu groß -> Toleranzfenster für Kanäle einstellen. Kanalverdrahtung und Sensorkonfiguration prüfen. |  |  | 值差异过大 -> 调整通道的容差范围. 检查通道接线和传感器配置.
  Err_524 | Stuck at error | Stuck at error | Hängengeblieben bei Fehler |  |  | 卡在错误处
  Err_525 | Readback error -> Check I/O module wiring. Restart I/O module, if needed. If this error persists, replace I/O module. | Readback error -> Check I/O module wiring. Restart I/O module, if needed. If this error persists, replace I/O module. | Fehler Rücklesen -> Verdrahtung des E/A-Moduls überprüfen. Bei Bedarf E/A-Modul neu starten. Falls der Fehler weiterhin besteht, E/A-Modul austauschen. |  |  | 回读错误 -> 检查 I/O 模块接线. 如果需要，重新启动 I/O 模块. 如果此错误仍然存在，请更换 I/O 模块.
  Err_530 | Class 3: Cross-talk error; Class 4: Internal fuse at 0V is defect. 0V not connected with GND -> Check I/O module wiring. Restart I/O module, if needed. If this error persists, replace I/O module. | Class 3: Cross-talk error; Class 4: Internal fuse at 0V is defect. 0V not connected with GND -> Check I/O module wiring. Restart I/O module, if needed. If this error persists, replace I/O module. | Klasse 3: Fehler Kanalübersprechen; Klasse 4: Interne Sicherung an 0 V defekt. 0 V nicht an GND angeschlossen -> Verdrahtung des E/A-Moduls überprüfen. Bei Bedarf E/A-Modul neu starten. Falls der Fehler weiterhin besteht, E/A-Modul austauschen. |  |  | 3 级：串扰错误; 4 级：0V 时内部保险丝有缺陷. 0V 未连接 GND -> 检查 I/O 模块接线. 如果需要，重新启动 I/O 模块. 如果此错误仍然存在，请更换 I/O 模块.
  Err_540 | Test error | Test error | Testfehler |  |  | 测试错误
  Err_555 | Internal error | Internal error | Interner Fehler |  |  | 内部错误
  Err_559 | Short circuit at digital output -> Check channel wiring | Short circuit at digital output -> Check channel wiring | Kurzschluss an Digitalausgang -> Kanalverdrahtung prüfen |  |  | 数字输出端短路 -> 检查通道接线
  Err_772 | Measurement overflow -> Check channel wiring | Measurement overflow -> Check channel wiring | Messwertüberschreitung -> Kanalverdrahtung prüfen |  |  | 测量值溢出 -> 检查通道接线
  Err_775 | Measurement underflow at analog input -> Check channel wiring | Measurement underflow at analog input -> Check channel wiring | Messwertunterschreitung an Analogausgang -> Kanalverdrahtung prüfen |  |  | 模拟输入端测量值下溢 -> 检查通道接线
  Err_796 | Different configuration | Different configuration | Abweichende Konfiguration |  |  | 配置不同
  Err_8480 | Not supported protocol variant | Not supported protocol variant | Nicht unterstützte Protokollvariante |  |  | 不支持的协议变体
  Err_8482 | Class 2: Timeout while initializing; Class 4: Timeout while waiting for ready status | Class 2: Timeout while initializing; Class 4: Timeout while waiting for ready status | Klasse 2: Timeout bei Initialisierung; Klasse 4: Timeout beim Warten auf Status „Bereit“ |  |  | 2 级：初始化超时; 4 级：等待就绪状态超时
  Err_8483 | Timeout during parameterization | Timeout during parameterization | Timeout bei Parametrierung |  |  | 参数化期间超时
  Err_8707 | PROFIsafe watchdog timed out | PROFIsafe watchdog timed out | Timeout von PROFIsafe-Watchdog |  |  | PROFIsafe 看门狗超时
  Err_8708 | Overvoltage | Overvoltage | Überspannung |  |  | 过电压
  Err_8711 | Undervoltage | Undervoltage | Unterspannung |  |  | 欠电压
  Err_8722 | Internal error | Internal error | Interner Fehler |  |  | 内部错误
  Err_8723 | Checksum error has occured in iParameters | Checksum error has occured in iParameters | Prüfsummenfehler in iParameter |  |  | i 参数中出现校验和错误
  Err_8724 | PROFIsafe communication error | PROFIsafe communication error | PROFIsafe-Kommunikationsfehler |  |  | PROFIsafe 通信错误
  Err_8732 | Internal error | Internal error | Interner Fehler |  |  | 内部错误
  Err_8747 | Internal runtime error | Internal runtime error | Interner Laufzeitfehler |  |  | 内部运行时错误
  Err_8961 | Wrong parameter value, check configuration | Wrong parameter value, check configuration | Falscher Parameterwert, Konfiguration prüfen |  |  | 参数值错误，请检查配置
  Err_8979 | Checksum error has occured in iParameter or F-Parameters | Checksum error has occured in iParameter or F-Parameters | Prüfsummenfehler in iParameter oder F-Parametern |  |  | i 参数或 F 参数中出现校验和错误
  Err_8986 | Invalid configuration -> Check modules and parameterization | Invalid configuration -> Check modules and parameterization | Ungültige Konfiguration -> Module und Parametrierung prüfen |  |  | 配置无效 -> 检查模块和参数化
  Err_8988 | F-Parameter configuration and address switch value do not match -> Check I/O module F-Parameter configuration and module address switch value. | F-Parameter configuration and address switch value do not match -> Check I/O module F-Parameter configuration and module address switch value. | Konfiguration für F-Parameter und Wert des Adressschalters stimmen nicht überein -> Konfiguration für F-Parameter des E/A-Moduls und Wert des Adressschalters überprüfen. |  |  | F 参数配置和地址开关值不匹配 -> 检查 I/O 模块 F 参数配置和模块地址开关值.
  Err_9249 | Timeout while waiting for Reset | Timeout while waiting for Reset | Timeout beim Warten auf Zurücksetzen |  |  | 等待重置时超时
  Err_9258 | Breakdown, communication lost | Breakdown, communication lost | Ausfall, Kommunikation unterbrochen |  |  | 故障，通信中断
  Err_9480 | I/O module removed from hotswap terminal unit or defective module on hotswap terminal unit -> Plug I/O module, replace I/O module | I/O module removed from hotswap terminal unit or defective module on hotswap terminal unit -> Plug I/O module, replace I/O module | E/A-Modul von Hotswap-Terminal-Einheit entfernt oder defektes Modul an Hotswap-Terminal-Einheit -> E/A-Modul einstecken, E/A-Modul austauschen |  |  | I/O 模块已从热插拔终端单元上拔下，或热插拔终端单元上的模块有故障 -> 插入 I/O 模块，更换 I/O 模块
  Err_9500 | Wrong I/O module plugged on hotswap terminal unit -> Remove wrong I/O module and plug projected I/O module | Wrong I/O module plugged on hotswap terminal unit -> Remove wrong I/O module and plug projected I/O module | Falsches E/A-Modul an Hotwwap-Terminal-Einheit eingesteckt -> Falsches E/A-Modul entfernen oder projektiertes E/A-Modul einstecken |  |  | 热插拔终端单元上插入了错误的 I/O 模块 -> 拔出错误的 I/O 模块并插入预计的 I/O 模块
  Err_9514 | No communication with I/O module on hotswap terminal unit -> Replace I/O module | No communication with I/O module on hotswap terminal unit -> Replace I/O module | Keine Kommunikation mit E/A-Modul an Hotswap-Terminal-Einheit -> E/A-Modul austauschen |  |  | 无法与热插拔终端单元上的 I/O 模块通信 -> 更换 I/O 模块
  Err_9526 | I/O module does not support hotswap functionality -> Power off system and replace I/O module | I/O module does not support hotswap functionality -> Power off system and replace I/O module | E/A-Modul unterstützt keine Hotswap-Funktion -> System abschalten und E/A-Modul austauschen |  |  | I/O 模块不支持热插拔功能 -> 关闭系统电源并更换 I/O 模块
  Err_9736 | hotswap terminal unit required but not found | hotswap terminal unit required but not found | Hotswap-Terminal-Einheit erforderlich, jedoch nicht gefunden |  |  | 需要热插拔终端单元但未找到
  Err_9764 | Defective hotswap terminal unit | Defective hotswap terminal unit | Defekte Hotswap-Terminal-Einheit |  |  | 热插拔终端单元有缺陷
  Err_9770 | No communication with hotswap terminal unit -> Restart, if error persists replace terminal unit | No communication with hotswap terminal unit -> Restart, if error persists replace terminal unit | Keine Kommunikation mit Hotswap-Terminal-Einheit -> Neu starten, falls Fehler weiterhin besteht, Terminal-Einheit austauschen |  |  | 无法与热插拔终端单元通信 -> 重新启动，如果错误仍然存在，请更换终端单元
  Hwd_14 | I/O bus | I/O bus | E/A-Bus |  |  | I/O 总线
  Sub1_ | Module | Module | Modul |  |  | 模块
  Sub2_ | Channel | Channel | Kanal |  |  | 通道
   |  |  |  |  |  |  *)

(* text list Diag_V3_PLC (id | default | en | de | fr | es | zh)
  Add_570425344 | Unknown reason | Unknown reason | Unbekannter Fehler |  |  | 未知原因
  Add_570425345 | Shutdown of the PLC | Shutdown of the PLC | Abschaltung der SPS |  |  | 关闭 PLC
  Add_570425346 | Reset after having stopped the IEC application | Reset after having stopped the IEC application | Nach Stoppen der IEC-Anwendung zurücksetzen |  |  | 在停止 IEC 应用程序后重置
  Add_570425347 | Exception occurred | Exception occurred | Ausnahme aufgetreten |  |  | 发生异常
  Add_570425348 | IEC application stopped by user | IEC application stopped by user | IEC-Anwendung durch Benutzer gestoppt |  |  | IEC 应用程序由用户停止
  Add_570425349 | IEC application stopped by function block | IEC application stopped by function block | IEC-Anwendung durch Funktionsbaustein gestoppt |  |  | IEC 应用程序由功能块停止
  Add_570425350 | IEC application will be deleted after the stop | IEC application will be deleted after the stop | IEC-Anwendung wird nach Stopp gelöscht |  |  | IEC 应用程序将在停止后被删除
  Add_570425351 | IEC application stopped because of debugging | IEC application stopped because of debugging | IEC-Anwendung wegen Debugging gestoppt |  |  | IEC 应用程序因调试而停止
  Add_570425352 | IEC application stopped because the run stop switch is on stop | IEC application stopped because the run stop switch is on stop | IEC-Anwendung wurde gestoppt, da Laufstopp-Schalter auf „Stopp“ gesetzt ist |  |  | IEC 应用程序因运行停止开关处于停止位置而停止
  Add_587202560 | Reset warm | Reset warm | Zurücksetzen (warm) |  |  | 热重置
  Add_587202561 | Reset cold | Reset cold | Zurücksetzen (kalt) |  |  | 冷重置
  Add_587202562 | Reset origin | Reset origin | Zurücksetzen (Original) |  |  | 重置原点
  Add_587202563 | Reset device | Reset device | Gerät zurücksetzen |  |  | 重置设备
  Add_637534224 | Software watchdog of IEC task expired | Software watchdog of IEC task expired | Software-Watchdog von IEC-Aufgabe abgelaufen |  |  | IEC 任务的软件看门狗已过期
  Add_637534225 | Hardware watchdog expired. Global software error | Hardware watchdog expired. Global software error | Hardware-Watchdog abgelaufen. Globaler Software-Fehler |  |  | 硬件看门狗已过期. 全局软件错误
  Add_637534226 | I/O configuration error | I/O configuration error | E/A-Konfigurationsfehler |  |  | I/O 配置错误
  Add_637534227 | Checksum error after program download | Checksum error after program download | Prüfsummenfehler nach Programm-Download |  |  | 程序下载后校验和错误
  Add_637534228 | Fieldbus error | Fieldbus error | Feldbus-Fehler |  |  | Fieldbus 错误
  Add_637534229 | I/O update error | I/O update error | E/A-Update-Fehler |  |  | I/O 更新错误
  Add_637534230 | Cycle time exceeded | Cycle time exceeded | Zykluszeit überschritten |  |  | 已超出循环时间
  Add_637534231 | Program too large for online change | Program too large for online change | Programm zu groß für Online-Änderung |  |  | 程序过大，无法在线更改
  Add_637534232 | Unresolved external references | Unresolved external references | Nicht aufgelöste externe Referenzen |  |  | 未解决的外部引用
  Add_637534233 | Download was rejected | Download was rejected | Download abgelehnt |  |  | 下载被拒绝
  Add_637534234 | Boot project not loaded because retain variables could not be relocated | Boot project not loaded because retain variables could not be relocated | Boot-Projekt nicht geladen, da Retain-Variablen nicht geladen werden konnten |  |  | 由于保留变量无法重定位，引导项目未加载
  Add_637534235 | Boot project not loaded and deleted | Boot project not loaded and deleted | Boot-Projekt nicht geladen und gelöscht |  |  | 引导项目未加载且已删除
  Add_637534236 | Out of heap memory | Out of heap memory | Kein Heap-Speicher mehr verfügbar |  |  | 堆内存不足
  Add_637534237 | Retain memory corrupt or cannot be mapped | Retain memory corrupt or cannot be mapped | Retain-Speicher beschädigt oder kann nicht zugeordnet werden |  |  | 保留内存损坏或无法映射
  Add_637534238 | Boot project could be loaded but caused an exception | Boot project could be loaded but caused an exception | Boot-Projekt konnte aufgrund einer Ausnahme nicht geladen werden |  |  | 引导项目可以加载，但会导致异常
  Add_637534241 | Target of the boot project doesn't match the current target | Target of the boot project doesn't match the current target | Ziel von Boot-Projekt stimmt nicht mit aktuellem Ziel überein |  |  | 引导项目的目标与当前目标不匹配
  Add_637534242 | Error at scheduling IEC tasks | Error at scheduling IEC tasks | Fehler bei der Zeitplanung von IEC-Aufgaben |  |  | 安排 IEC 任务时出错
  Add_637534243 | Checksum of downloaded file does not match | Checksum of downloaded file does not match | Diskrepanz bei Prüfsumme der heruntergeladenen Datei |  |  | 下载文件的校验和不匹配
  Add_637534244 | Retain identity does not match to current boot application program identity | Retain identity does not match to current boot application program identity | Retain-Identität stimmt nicht mit aktueller Identität des Boot-Anwendungsprogramms überein |  |  | 保留标识与当前引导应用程序标识不匹配
  Add_637534245 | IEC task configuration failed | IEC task configuration failed | IEC-Aufgabenkonfiguration fehlgeschlagen |  |  | IEC 任务配置失败
  Add_637534246 | Application is running on wrong target. Can be used for library protection! | Application is running on wrong target. Can be used for library protection! | Anwendung läuft über falsches Ziel. Kann zum Schutz der Bibliothek verwendet werden! |  |  | 应用程序在错误的目标上运行. 可用于库保护！
  Add_637534288 | Illegal instruction | Illegal instruction | Ungültige Anweisung |  |  | 非法指令
  Add_637534289 | Access violation | Access violation | Zugriffsverletzung |  |  | 访问冲突
  Add_637534290 | Privileged instruction | Privileged instruction | Privilegierte Anweisung |  |  | 特权指令
  Add_637534292 | Stack overflow | Stack overflow | Stack-Überlauf |  |  | 堆栈溢出
  Add_637534293 | Invalid disposition | Invalid disposition | Ungültige Löschung |  |  | 处置无效
  Add_637534294 | Invalid handle | Invalid handle | Ungültiger Handle |  |  | 句柄无效
  Add_637534295 | Guard page | Guard page | Guard-Seite |  |  | 守护页面
  Add_637534296 | Double fault | Double fault | Doppelfehler |  |  | 双重故障
  Add_637534297 | Invalid OpCode | Invalid OpCode | Ungültiger OpCode |  |  | 操作码无效
  Add_637534464 | Data type misalignment | Data type misalignment | Abweichender Datentyp |  |  | 数据类型不一致
  Add_637534465 | Array bounds exceeded | Array bounds exceeded | Array-Grenzen überschritten |  |  | 超出数组边界
  Add_637534466 | Division by zero | Division by zero | Division durch Null |  |  | 除以零
  Add_637534467 | Overflow | Overflow | Überlauf |  |  | 溢出
  Add_637534468 | Non continuable | Non continuable | Nicht fortführbar |  |  | 非连续性
  Add_637534469 | Processor load watchdog of all IEC tasks detected | Processor load watchdog of all IEC tasks detected | Prozessorlast-Watchdog aller IEC-Aufgaben erkannt |  |  | 检测到所有 IEC 任务的处理器负载看门狗
  Add_637534544 | FPU: Unspecified error | FPU: Unspecified error | FPU: Nicht spezifizierter Fehler |  |  | FPU：不明错误
  Add_637534545 | FPU: Denormalized operand | FPU: Denormalized operand | FPU: Denormalisierter Operand |  |  | FPU：非规范化操作数
  Add_637534546 | FPU: Division by zero | FPU: Division by zero | FPU: Division durch Null |  |  | FPU：除以零
  Add_637534547 | FPU: Inexact result | FPU: Inexact result | FPU: Ungenaues Ergebnis |  |  | FPU：结果不准确
  Add_637534548 | FPU: Invalid operation | FPU: Invalid operation | FPU: Ungültige Operation |  |  | FPU：无效操作
  Add_637534549 | FPU: Overflow | FPU: Overflow | FPU: Überlauf |  |  | FPU：溢出
  Add_637534550 | FPU: Stack check | FPU: Stack check | FPU: Stack-Prüfung |  |  | FPU：堆栈检查
  Add_637534551 | FPU: Underflow | FPU: Underflow | FPU: Unterlauf |  |  | FPU：下溢
  Add_637534720 | Hardware breakpoint | Hardware breakpoint | Hardware-Breakpoint |  |  | 硬件断点
  Add_637538320 | Omitted cycle watchdog | Omitted cycle watchdog | Zyklus-Watchdog ausgelassen |  |  | 已省略循环看门狗
  Err_10 | Medium has almost used its complete spare capacity or is already dead, action required | Medium has almost used its complete spare capacity or is already dead, action required | Fast die gesamte freie Kapazität des Mediums ist belegt oder es ist bereits deaktiviert, Maßnahme erforderlich |  |  | 介质的全部备用容量已经接近用尽或已经用尽，需要采取措施
  Err_11 | Type scaling on PLC startup failed | Type scaling on PLC startup failed | Typskalierung bei SPS-Start fehlgeschlagen |  |  | PLC 启动时的类型扩展失败
  Err_12 | Flash is temporary protected (read only) | Flash is temporary protected (read only) | Flash-Speicher ist temporär geschützt (schreibgeschützt) |  |  | 闪存受到临时保护（只读）
  Err_17 | Error setting parameters | Error setting parameters | Fehlereinstellungsparameter |  |  | 设置参数时出错
  Err_18 | At least one not found | At least one not found | Mindestens eine/r/s nicht gefunden |  |  | 至少有一个未找到
  Err_19 | Unable to read at least one value | Unable to read at least one value | Lesen von mindestens einem Fehler fehlgeschlagen |  |  | 无法读取至少一个值
  Err_2 | Resource failure | Resource failure | Ressourcenfehler |  |  | 资源故障
  Err_20 | Invalid value of "Error LED" | Invalid value of "Error LED" | Ungültiger Wert für „Fehler-LED“ |  |  | “错误 LED”的值无效
  Err_21 | Invalid value of "Check battery" | Invalid value of "Check battery" | Ungültiger Wert für „Überwachung Batteriestatus“ |  |  | “检查电池”的值无效
  Err_22 | Error at initialization | Error at initialization | Fehler bei der Initialisierung |  |  | 初始化时出错
  Err_23 | Wrong version of firmware | Wrong version of firmware | Falsche Firmware-Version |  |  | 固件版本错误
  Err_24 | Invalid value of parameter "Diagnosis, stop on error class" | Invalid value of parameter "Diagnosis, stop on error class" | Ungültiger Wert für Parameter „Diagnose, Stopp bei Fehlerklasse“ |  |  | 参数“诊断，出现错误类别时停止”的值无效
  Err_25 | Invalid value of parameter "Diagnosis, add Plc name to node name" | Invalid value of parameter "Diagnosis, add Plc name to node name" | Ungültiger Wert für Parameter „Diagnose, SPS-Namen zum Knotennamen hinzufügen“ |  |  | 参数“诊断，将 PLC 名称添加到节点名称”的值无效
  Err_26 | Invalid value of parameter "Reboot at powerfail" | Invalid value of parameter "Reboot at powerfail" | Ungültiger Wert für Parameter „Bei Stromausfall neu starten“ |  |  | 参数“电源故障时重新引导”的值无效
  Err_27 | Failed to set parameter "Reboot at powerfail" | Failed to set parameter "Reboot at powerfail" | Einstellen von Parameter „Bei Stromausfall neu starten“ fehlgeschlagen |  |  | 无法设置参数“电源故障时重新引导”
  Err_28 | Value of parameter "Missed Cycle Task behaviour" is not in range | Value of parameter "Missed Cycle Task behaviour" is not in range | Wert von Parameter „Verhalten bei versäumter Zyklusaufgabe“ liegt außerhalb des zulässigen Bereichs |  |  | 参数“错过周期任务行为”的值不在范围内
  Err_29 | Combination of plugged option boards is invalid | Combination of plugged option boards is invalid | Kombination von eingesteckten Optionskarten ist ungültig |  |  | 插入的选项板组合无效
  Err_3 | Timeout | Timeout | Timeout |  |  | 超时
  Err_30 | Value of parameter "Priority Scheme" is not in range | Value of parameter "Priority Scheme" is not in range | Wert von Parameter „Prioritätsschema“ liegt außerhalb des zulässigen Bereichs |  |  | 参数“优先级方案”的值不在范围内
  Err_31 | PLC did not go to RUN mode due to an active error, whose severity exceeds value of parameter 'stop on error class' | PLC did not go to RUN mode due to an active error, whose severity exceeds value of parameter 'stop on error class' | SPS ist aufgrund eines aktiven Fehlers, dessen Schweregrad den Wert für Parameter „Stoppen bei Fehlerklasse“ überschreitet, nicht in den RUN-Modus gewechselt |  |  | 由于存在严重程度超出“出错时停止类”参数值的活动错误，PLC 未进入运行模式。
  Err_32 | PLC went to STOP mode due to occurence of an error, whose severity exceeds value of parameter 'stop on error class' | PLC went to STOP mode due to occurence of an error, whose severity exceeds value of parameter 'stop on error class' | SPS ist aufgrund eines Fehlers, dessen Schweregrad den Wert für Parameter „Stoppen bei Fehlerklasse“ überschreitet, in den STOPP-Modus gewechselt |  |  | 由于发生严重程度超出“出错时停止类”参数值的错误，PLC 进入停止模式。
  Err_33 | PLC went to RUN mode | PLC went to RUN mode | SPS in RUN-Modus gewechselt |  |  | PLC 进入运行模式
  Err_34 | PLC went to STOP mode | PLC went to STOP mode | SPS in STOPP-Modus gewechselt |  |  | PLC 进入停止模式
  Err_35 | IEC application has been reset | IEC application has been reset | IEC-Anwendung wurde zurückgesetzt |  |  | IEC 应用程序已重置
  Err_36 | Online change of IEC application has been performed | Online change of IEC application has been performed | Online-Änderung von IEC-Anwendung wurde vorgenommen |  |  | 已执行 IEC 应用程序的在线更改
  Err_37 | Full download of an IEC application has been performed | Full download of an IEC application has been performed | Vollständiger Download einer IEC-Anwendung wurde ausgeführt |  |  | 已执行 IEC 应用程序的完整下载
  Err_38 | IEC application caused an exception | IEC application caused an exception | IEC-Anwendung hat eine Ausnahme verursacht |  |  | IEC 应用程序导致异常
  Err_39 | PLC did not go to RUN mode since reboot has to be performed first | PLC did not go to RUN mode since reboot has to be performed first | SPS ist nicht in den RUN-Modus gewechselt, da zunächst Neustart ausgeführt werden musste |  |  | PLC 未进入运行模式，必须先执行重新引导
  Err_40 | Value of parameter "Reboot on E2" is not in range | Value of parameter "Reboot on E2" is not in range | Wert von Parameter „Neu starten bei E2“ liegt außerhalb des zulässigen Bereichs |  |  | 参数“在 E2 时重新引导”的值不在范围内
  Err_41 | PLC went to reboot due to occurence of an E2 error | PLC went to reboot due to occurence of an E2 error | SPS ist aufgrund eines E2-Fehlers neu gestartet |  |  | 由于发生 E2 错误，PLC 重新引导
  Err_42 | No boot project loaded | No boot project loaded | Kein Boot-Projekt geladen |  |  | 引导项目未加载
  Err_43 | Boot project loaded | Boot project loaded | Boot-Projekt geladen |  |  | 引导项目已加载
  Err_44 | Loading boot project failed due to failing load of retain data | Loading boot project failed due to failing load of retain data | Laden von Boot-Projekt aufgrund von Fehler beim Laden von Retain-Daten fehlgeschlagen |  |  | 由于保留数据加载失败，引导项目加载失败
  Err_45 | Loading boot project failed due to mismatch of retain data | Loading boot project failed due to mismatch of retain data | Laden von Boot-Projekt aufgrund einer Diskrepanz der Retain-Daten fehlgeschlagen |  |  | 由于保留数据不匹配，引导项目加载失败
  Err_46 | Loading boot project failed due to insufficient license for application | Loading boot project failed due to insufficient license for application | Laden von Boot-Projekt aufgrund einer unzureichenden Anwendungslizenz fehlgeschlagen |  |  | 由于应用程序许可证不足，引导项目加载失败
  Err_47 | Loading boot project failed due to unspecified reason | Loading boot project failed due to unspecified reason | Laden von Boot-Projekt aus unbekanntem Grund fehlgeschlagen |  |  | 由于不明原因，引导项目加载失败
  Err_48 | Backup failed | Backup failed | Backup fehlgeschlagen |  |  | 备份失败
  Err_49 | Restore failed | Restore failed | Wiederherstellung fehlgeschlagen |  |  | 还原失败
  Err_50 | Invalid value of parameter "Enable diagnosis history" | Invalid value of parameter "Enable diagnosis history" | Ungültiger Wert für Parameter „Diagnosehistorie aktivieren“ |  |  | 参数“启用诊断历史记录”的值无效
  Err_51 | Invalid value of parameter "Maximum number of entries in diagnosis history" | Invalid value of parameter "Maximum number of entries in diagnosis history" | Ungültiger Wert für Parameter „Maximale Anzahl von Einträgen in Diagnosehistorie“ |  |  | 参数“诊断历史记录中的最大条目数”的值无效
  Err_52 | Invalid value of parameter "Maximum size of extended diagnosis data in diagnosis history" | Invalid value of parameter "Maximum size of extended diagnosis data in diagnosis history" | Ungültiger Wert für Parameter „Maximale Größe von erweiterten Diagnosedaten in Diagnosehistorie“ |  |  | 参数“诊断历史记录中扩展诊断数据的最大大小”的值无效
  Err_53 | System partition free space has fallen below pre-warn threshold -> Please contact your ABB representative to fix this issue | System partition free space has fallen below pre-warn threshold -> Please contact your ABB representative to fix this issue | Freier Speicherplatz der Systempartition ist unter Vorwarngrenze gesunken -> Zur Behebung dieses Problems entsprechenden ABB-Vertreter kontaktieren |  |  | 系统分区可用空间已降至低于预警阈值 -> 请联系您的 ABB 代表以解决此问题
  Err_54 | System Partition has run out of space -> Please contact your ABB representative to fix this issue and replace the CPU as soon as possible | System Partition has run out of space -> Please contact your ABB representative to fix this issue and replace the CPU as soon as possible | Systempartition hat keinen Speicherplatz mehr -> Zur Behebung dieses Problems entsprechenden ABB-Vertreter kontaktieren und schnellstmöglich CPU austauschen |  |  | 系统分区空间已用尽 -> 请联系您的 ABB 代表以解决此问题，并且尽快更换 CPU
  Err_55 | IEC project prevented from going to RUN mode, see PLC log for details | IEC project prevented from going to RUN mode, see PLC log for details |  |  |  | 
  Err_8 | Empty or missing | Empty or missing | Leer oder fehlt |  |  | 空或缺失
  Err_9 | Medium has used 80% of its spare capacity | Medium has used 80% of its spare capacity | 80 % der freien Kapazität von Medium belegt |  |  | 介质的备用容量已经使用 80%
  Hwd_0 | CPU | CPU | CPU |  |  | CPU
  Sub1_0 | CPU | CPU | CPU |  |  | CPU
  Sub1_14 | I/O bus | I/O bus | E/A-Bus |  |  | I/O 总线
  Sub1_19 | Flashdisk | Flashdisk | Flashdisk |  |  | 闪盘
  Sub1_21 | Display | Display | Anzeige |  |  | 显示
  Sub1_22 | Battery | Battery | Batterie |  |  | 电池
  Sub2_0 | Device | Device | Gerät |  |  | 设备
  Sub2_2 | Parameter | Parameter | Parameter |  |  | 参数
  Sub2_5 | Index | Index | Index |  |  | 索引
  Sub2_6 | Application | Application | Anwendung |  |  | 应用程序
  Sub2_7 | Bootproject | Bootproject |  |  |  | 
  Sub2_8 | Component | Component |  |  |  | 
  Sub4_1 | too big | too big | zu groß |  |  | 过大
  Sub4_2 | too small | too small | zu klein |  |  | 过小
  Sub4_3 | unequal | unequal | ungleich |  |  | 不等于
  Sub4_4 | equal | equal | gleich |  |  | 等于
   |  |  |  |  |  |  *)
